// TIA Portal V20 export
// export: Created 2025-12-01T14:56:34.3256321Z, ExportSetting None, DisplayName Totally Integrated Automation Portal, DisplayVersion V20 Update 3, DisplayName TIA Portal Openness, DisplayVersion V20 Update 3, DisplayName TIA Portal Version Control Interface, DisplayVersion V20 Update 3, DisplayName STEP 7 Professional, DisplayVersion V20 Update 3, DisplayName STEP 7 Safety, DisplayVersion V20 Update 2, DisplayName WinCC Basic/Comfort/Advanced, DisplayVersion V20 Update 3, DisplayName WinCC Professional, DisplayVersion V20 Update 3, DisplayName WinCC Unified, DisplayVersion V20 Update 3
FUNCTION_BLOCK "FB463_CRTL_TR_TP_E1E2_S234_Pres"   // FB463, LAD
TITLE = bimba y lola
{ S7_Optimized_Access := 'FALSE' }
AUTHOR : TLigero
NAME : 20180827
VERSION : 3.0
// pendiente de simular
// stored: AutoNumber false, SetENOAutomatically false
   VAR_INPUT
      Mesa : UInt;   // Número de mesa
      En_Tension : Bool;
      pHsMx : Bool;   // pHs de presencia de la Mesa
      TP1_Up : Bool;   // TP1 Arriba. E1 >> S3. si no hay tope poner ON
      TP1_Down : Bool;   // TP1 Abajo. E1 >> S3. si no hay tope poner ON
      PosTR_E1 : Bool;   // Posicion del TR en E1E3
      PosTR_E2 : Bool;   // Posicion del TR en E2E4
      Termico_13 : Bool;   // Proteccion del Tx en E1E3
      Termico_24 : Bool;   // Proteccion del Tx en E2E4
      Avance_13 : Bool;   // Avance del Tx en E1E3
      Avance_24 : Bool;   // Avance del Tx en E2E4
      Retroceso_24 : Bool;   // Retroceso del Tx en E2E4
      PTF_Sal_M2 : Bool;   // S2 >> Mesa Siguiente PTF
      NXT_Avance_S2 : Bool;   // S2 >> Mesa Siguiente avanzando
      PTF_Sal_M3 : Bool;   // S3 >> Mesa Siguiente PTF
      NXT_Avance_S3 : Bool;   // S3 >> Mesa Siguiente avanzando
      PTF_Sal_M4 : Bool;   // S4 >> Mesa Siguiente PTF
      NXT_Avance_S4 : Bool;   // S4 >> Mesa Siguiente avanzando
      F_EnvMens_Mx : Bool;   // Fin de Envio de Mensaje
      Mx_Bloq_Activo : Bool;   // Bloqueo Activo de la Mesa
      Mx_FlujoPrin_S2 : Bool;   // para flujo principal S3 dejar los dos flujos principales a off
      Mx_FlujoPrin_S4 : Bool;   // para flujo principal S3 dejar los dos flujos principales a off
      AVTF_Ent_M1 : Bool;   // E1 >> Mesa Anterior AVTF
      AVTF_Ent_M2 : Bool;   // E2 >> Mesa Anterior AVTF
      Num_Cruce : UInt;   // Número de cruce.
      DB_FIFO_Cruce : UInt := 213;   // DB de la FIFO de ordenes del cruce
      Long_FIFO_Cruce : UInt := 1;   // Longitut de la FIFO de ordenes del cruce
      ValorOrden_S2 : Word := 16#81;   // Con que orden entra por S2
      ValorOrden_S4 : Word := 16#82;   // Con que orden entra por S4
      MesaS2 : UInt;   // Número de mesa por S2
      MesaS3 : UInt;   // Número de mesa por S3
      MesaS4 : UInt;   // Número de mesa por S4
      V_CNT_pHsMx_E1 : UDInt := 500;   // Valor de presencia por E1 en ms
      V_CNT_pHsMx_E2 : UDInt := 500;   // Valor de presencia por E2 en ms
      V_CNT_ApHsMx_S2 : UDInt := 500;   // Valor de Ausencia por S2 en ms
      V_CNT_ApHsMx_S3 : UDInt := 500;   // Valor de Ausencia por S3 en ms
      V_CNT_ApHsMx_S4 : UDInt := 500;   // Valor de Ausencia por S4 en ms
      V_TOut_Tx_Mx : UDInt := 3000;   // TimeOut de Atasco en ms
      V_TOut_TP : UDInt := 2000;   // TimeOut de Tope en ms
      V_TOut_TR : UDInt := 2000;   // TimeOut de Transfer en ms
      V_Paro : UDInt := 5000;   // tiempo que avanza el transportador sin aviso hasta que se para (ms)
      V_Vaciado : UDInt := 5000;   // Valor de vaciado en ms
   END_VAR
   VAR_OUTPUT
      P_EnvMens_PMx : Bool;   // Permiso de Enviar Mensaje de Presencia
      Etiqueta_Jdt : UDInt;   // Etiqueta que ha sido leida
      Orden_Ejecutada_Jdt : UInt;   // Orden que se ha ejecutado
      PTF_Ent_M1 : Bool;   // E1 >> Mesa Anterior PTF
      PTF_Ent_M2 : Bool;   // E2 >> Mesa Anterior PTF
      AVTF_Sal_M2 : Bool;   // S2 >> Mesa Siguiente AVTF
      NXT_Descarga_Act_S2 : Bool;   // S2 >> Mesa Siguiente descarga activa
      AVTF_Sal_M3 : Bool;   // S3 >> Mesa Siguiente AVTF
      NXT_Descarga_Act_S3 : Bool;   // S3 >> Mesa Siguiente descarga activa
      AVTF_Sal_M4 : Bool;   // S4 >> Mesa Siguiente AVTF
      NXT_Descarga_Act_S4 : Bool;   // S4 >> Mesa Siguiente descarga activa
   END_VAR
   VAR
      T1_ET00 : Bool;
      T1_ET01 : Bool;
      T1_ET02 : Bool;
      T1_ET03 : Bool;
      T1_ET10 : Bool;
      T1_ET11 : Bool;
      T1_ET20 : Bool;
      T1_ET21 : Bool;
      T1_ET50 : Bool;
      T1_ET60 : Bool;
      T1_ET80 : Bool;
      T1_ET110 : Bool;
      T1_ET111 : Bool;
      T1_ET112 : Bool;
      FIFO_OK : Bool;
      TRANS_OK : Bool;
      O_Bloqueo : Bool;
      Inv_sentido_24 : Bool;
      Ultima_entra_de_E2 : Bool;
      Ultima_entra_de_E1 : Bool;
      Err_Detec_PHS : Bool;
      Tim_Vaciado_Q : Bool;
      TMP_Atasco_Q : Bool;
      TMP_Paro_Q : Bool;
      FN_ET02 : Bool;
      Tmp_Tout_Tr_Q : Bool;
      TMP_Tout_tope_E2_Q : Bool;
      TMP_Tout_tope_E1_Q : Bool;
      maux_fp_disparo_e1 : Bool;
      maux_fp_disparo_e2 : Bool;
      TMP_pHs_E1 : UDInt;
      TMP_Aus_S2 : UDInt;
      TMP_Aus_S3 : UDInt;
      TMP_Aus_S4 : UDInt;
      CNT_pHs_E2 : UDInt;
      TIM_Vaciado : UDInt;
      TMP_Paro : UDInt;
      TMP_Tout_Tp_E2 : UDInt;
      TMP_Tout_Tp_E1 : UDInt;
      TMP_Tout_Tr : UDInt;
      TMP_Atasco : UDInt;
      TMP_En_tension : UDInt;
      Datos_Scanner { S7_SetPoint := 'True'} : "ROUT_Orden_Fifo_Scanner";
   END_VAR
   VAR_TEMP
      EstadoZona : "EstadoZona";   // Estado de Zona de la Mesa
      EstadoVI : "EstadosMesa";   // Estado del Vehiculo Inteliguente de la Mesa
      ConfigFB : "UDT_ConfigFB";   // Configuracion de la FB de la Mesa
      O_Sal_S2 : Bool;
      O_Sal_S4 : Bool;
      O_Sal_S3 : Bool;
      O_Vaciar : Bool;
      Moti_ERRO : Bool;
      Moti_NENC : Bool;
      Moti_NORM : Bool;
      Moti_INIC : Bool;
      tmp_Aus_S4_Q : Bool;
      tmp_pHs_E2_Q : Bool;
      tmp_pHs_E1_Q : Bool;
      tmp_pHs_S3_Q : Bool;
      tmp_pHs_S2_Q : Bool;
      ok_tension : Bool;
      Aux_W_Moti : Word;
      INT_ORDEN : UInt;
      Aux_W_Orden : Word;
      I_Ord_Filtrada : UInt;
      I_V_Ord_S4 : UInt;
      I_V_Ord_S2 : UInt;
   END_VAR
   VAR_TEMP   // added for the SCL form of the ladder/FBD networks
      _w1 : Bool;
      _w2 : Bool;
      _w3 : Bool;
      _w4 : Bool;
      _w5 : Bool;
      _w6 : Bool;
      _w7 : Bool;
   END_VAR
BEGIN

REGION Network 1: INICIALIZAR - Recoger las Variables de Estado de la Mesa
   // Se recoge - Estado_CBx
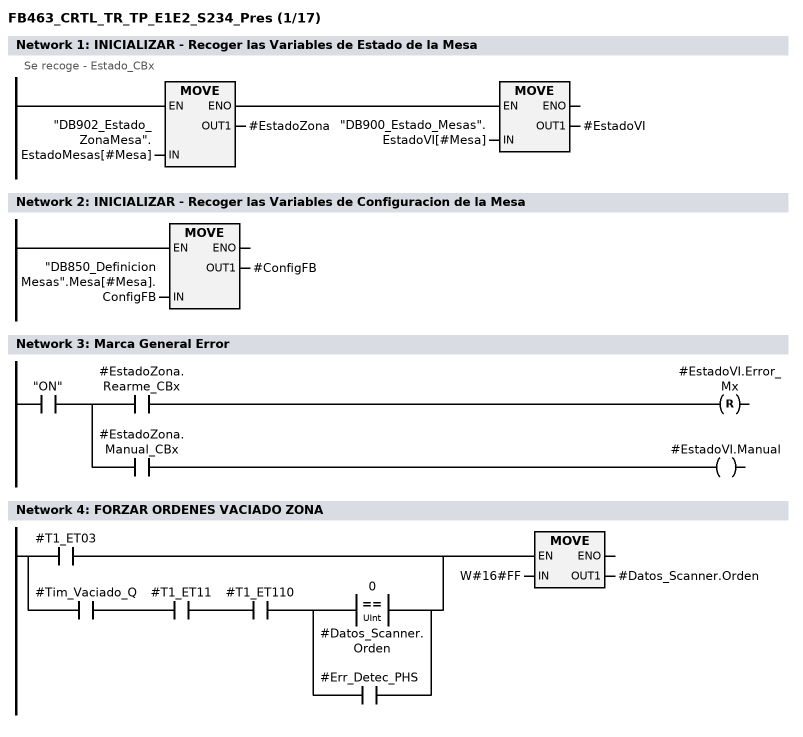
   RUNG wire#powerrail
      Move(in := "DB902_Estado_ZonaMesa".EstadoMesas[#Mesa], out1 => #EstadoZona)
      Move(in := "DB900_Estado_Mesas".EstadoVI[#Mesa], out1 => #EstadoVI)
   END_RUNG
   // the same network as SCL:
   #EstadoZona := "DB902_Estado_ZonaMesa".EstadoMesas[#Mesa];
   #EstadoVI := "DB900_Estado_Mesas".EstadoVI[#Mesa];
END_REGION

REGION Network 2: INICIALIZAR - Recoger las Variables de Configuracion de la Mesa
   RUNG wire#powerrail
      Move(in := "DB850_DefinicionMesas".Mesa[#Mesa].ConfigFB, out1 => #ConfigFB)
   END_RUNG
   // the same network as SCL:
   #ConfigFB := "DB850_DefinicionMesas".Mesa[#Mesa].ConfigFB;
END_REGION

REGION Network 3: Marca General Error
   RUNG wire#powerrail
      Contact( "ON" )
      wire#w1
      Contact( #EstadoZona.Rearme_CBx )
      R_Coil( #EstadoVI.Error_Mx )
   END_RUNG
   RUNG wire#w1
      Contact( #EstadoZona.Manual_CBx )
      Coil( #EstadoVI.Manual )
   END_RUNG
   // the same network as SCL:
   IF "ON" AND #EstadoZona.Rearme_CBx THEN #EstadoVI.Error_Mx := FALSE; END_IF;
   #EstadoVI.Manual := "ON" AND #EstadoZona.Manual_CBx;
END_REGION

REGION Network 4: FORZAR ORDENES VACIADO ZONA
   RUNG wire#powerrail
      Contact( #T1_ET03 )
      wire#w1
      { S7_GenerateENO := "TRUE" } Move(in := W#16#FF, out1 => #Datos_Scanner.Orden)
   END_RUNG
   RUNG wire#powerrail
      Contact( #Tim_Vaciado_Q )
      Contact( #T1_ET11 )
      Contact( #T1_ET110 )
      wire#w2
      { S7_Templates := "SrcType := UInt" } EQ_Contact(in1 := 0, in2 := #Datos_Scanner.Orden)
   END_RUNG wire#w1
   RUNG wire#w2
      Contact( #Err_Detec_PHS )
   END_RUNG wire#w1
   // the same network as SCL:
   IF #T1_ET03 OR (#Tim_Vaciado_Q AND #T1_ET11 AND #T1_ET110 AND ((0 = #Datos_Scanner.Orden) OR #Err_Detec_PHS)) THEN
       #Datos_Scanner.Orden := W#16#FF;
   END_IF;
END_REGION

REGION Network 5: evaluar la orden extraida de la fifo
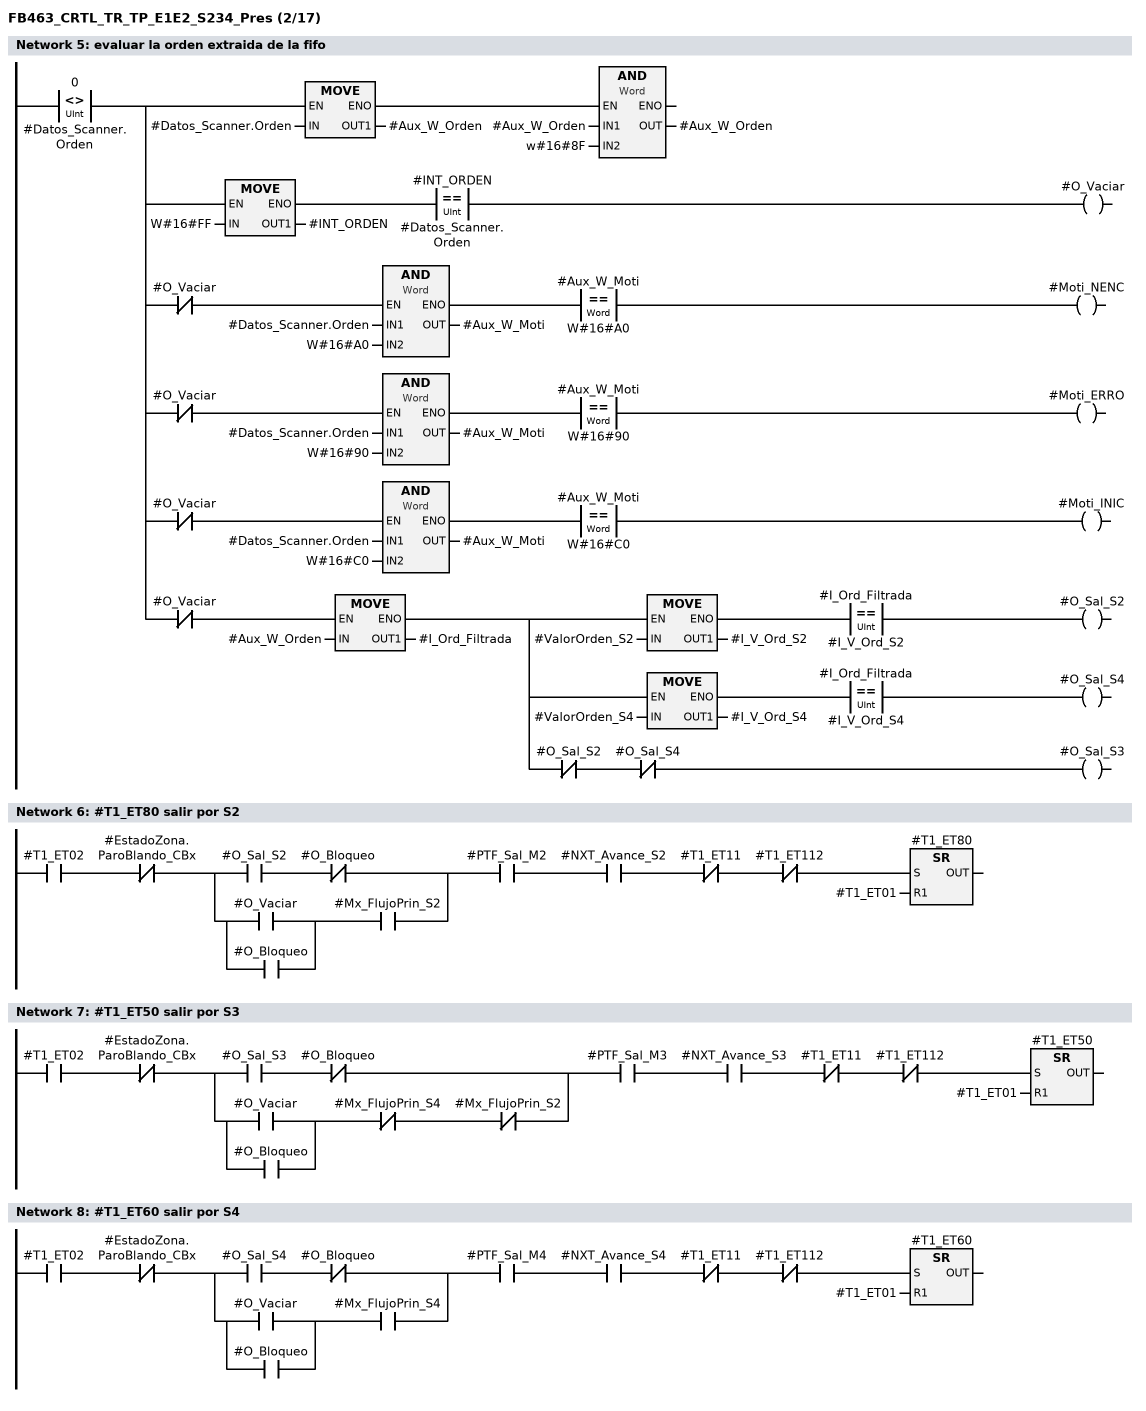
   RUNG wire#powerrail
      { S7_Templates := "SrcType := UInt" } NE_Contact(in1 := 0, in2 := #Datos_Scanner.Orden)
      wire#w1
      { S7_GenerateENO := "TRUE" } Move(in := #Datos_Scanner.Orden, out1 => #Aux_W_Orden)
      { S7_Templates := "SrcType := Word"; S7_GenerateENO := "TRUE" } And(in1 := #Aux_W_Orden, in2 := w#16#8F, out => #Aux_W_Orden)
   END_RUNG
   RUNG wire#w1
      { S7_GenerateENO := "TRUE" } Move(in := W#16#FF, out1 => #INT_ORDEN)
      { S7_Templates := "SrcType := UInt" } EQ_Contact(in1 := #INT_ORDEN, in2 := #Datos_Scanner.Orden)
      Coil( #O_Vaciar )
   END_RUNG
   RUNG wire#w1
      I_Contact( #O_Vaciar )
      { S7_Templates := "SrcType := Word"; S7_GenerateENO := "TRUE" } And(in1 := #Datos_Scanner.Orden, in2 := W#16#A0, out => #Aux_W_Moti)
      { S7_Templates := "SrcType := Word" } EQ_Contact(in1 := #Aux_W_Moti, in2 := W#16#A0)
      Coil( #Moti_NENC )
   END_RUNG
   RUNG wire#w1
      I_Contact( #O_Vaciar )
      { S7_Templates := "SrcType := Word"; S7_GenerateENO := "TRUE" } And(in1 := #Datos_Scanner.Orden, in2 := W#16#90, out => #Aux_W_Moti)
      { S7_Templates := "SrcType := Word" } EQ_Contact(in1 := #Aux_W_Moti, in2 := W#16#90)
      Coil( #Moti_ERRO )
   END_RUNG
   RUNG wire#w1
      I_Contact( #O_Vaciar )
      { S7_Templates := "SrcType := Word"; S7_GenerateENO := "TRUE" } And(in1 := #Datos_Scanner.Orden, in2 := W#16#C0, out => #Aux_W_Moti)
      { S7_Templates := "SrcType := Word" } EQ_Contact(in1 := #Aux_W_Moti, in2 := W#16#C0)
      Coil( #Moti_INIC )
   END_RUNG
   RUNG wire#w1
      I_Contact( #O_Vaciar )
      { S7_GenerateENO := "TRUE" } Move(in := #Aux_W_Orden, out1 => #I_Ord_Filtrada)
      wire#w2
      { S7_GenerateENO := "TRUE" } Move(in := #ValorOrden_S2, out1 => #I_V_Ord_S2)
      { S7_Templates := "SrcType := UInt" } EQ_Contact(in1 := #I_Ord_Filtrada, in2 := #I_V_Ord_S2)
      Coil( #O_Sal_S2 )
   END_RUNG
   RUNG wire#w2
      { S7_GenerateENO := "TRUE" } Move(in := #ValorOrden_S4, out1 => #I_V_Ord_S4)
      { S7_Templates := "SrcType := UInt" } EQ_Contact(in1 := #I_Ord_Filtrada, in2 := #I_V_Ord_S4)
      Coil( #O_Sal_S4 )
   END_RUNG
   RUNG wire#w2
      I_Contact( #O_Sal_S2 )
      I_Contact( #O_Sal_S4 )
      Coil( #O_Sal_S3 )
   END_RUNG
   // the same network as SCL:
   // ENO of a box is taken as its EN; it also drops when the box reports an error
   #_w1 := 0 <> #Datos_Scanner.Orden;
   IF #_w1 THEN
       #Aux_W_Orden := #Datos_Scanner.Orden;
       #Aux_W_Orden := #Aux_W_Orden AND w#16#8F;
       #INT_ORDEN := W#16#FF;
   END_IF;
   #O_Vaciar := #_w1 AND (#INT_ORDEN = #Datos_Scanner.Orden);
   #_w2 := #_w1 AND NOT #O_Vaciar;
   IF #_w2 THEN #Aux_W_Moti := #Datos_Scanner.Orden AND W#16#A0; END_IF;
   #Moti_NENC := #_w2 AND (#Aux_W_Moti = W#16#A0);
   #_w3 := #_w1 AND NOT #O_Vaciar;
   IF #_w3 THEN #Aux_W_Moti := #Datos_Scanner.Orden AND W#16#90; END_IF;
   #Moti_ERRO := #_w3 AND (#Aux_W_Moti = W#16#90);
   #_w4 := #_w1 AND NOT #O_Vaciar;
   IF #_w4 THEN #Aux_W_Moti := #Datos_Scanner.Orden AND W#16#C0; END_IF;
   #Moti_INIC := #_w4 AND (#Aux_W_Moti = W#16#C0);
   #_w5 := #_w1 AND NOT #O_Vaciar;
   IF #_w5 THEN
       #I_Ord_Filtrada := #Aux_W_Orden;
       #I_V_Ord_S2 := #ValorOrden_S2;
   END_IF;
   #O_Sal_S2 := #_w5 AND (#I_Ord_Filtrada = #I_V_Ord_S2);
   IF #_w5 THEN #I_V_Ord_S4 := #ValorOrden_S4; END_IF;
   #O_Sal_S4 := #_w5 AND (#I_Ord_Filtrada = #I_V_Ord_S4);
   #O_Sal_S3 := #_w5 AND NOT #O_Sal_S2 AND NOT #O_Sal_S4;
END_REGION

REGION Network 6: #T1_ET80 salir por S2
   RUNG wire#powerrail
      Contact( #T1_ET02 )
      I_Contact( #EstadoZona.ParoBlando_CBx )
      wire#w1
      Contact( #O_Sal_S2 )
      I_Contact( #O_Bloqueo )
      wire#w2
      Contact( #PTF_Sal_M2 )
      Contact( #NXT_Avance_S2 )
      I_Contact( #T1_ET11 )
      I_Contact( #T1_ET112 )
      S_SR(operand := #T1_ET80, r1 := #T1_ET01)
   END_RUNG
   RUNG wire#w1
      Contact( #O_Vaciar )
      wire#w3
      Contact( #Mx_FlujoPrin_S2 )
   END_RUNG wire#w2
   RUNG wire#w1
      Contact( #O_Bloqueo )
   END_RUNG wire#w3
   // the same network as SCL:
   IF #T1_ET02 AND NOT #EstadoZona.ParoBlando_CBx AND ((#O_Sal_S2 AND NOT #O_Bloqueo) OR ((#O_Vaciar OR #O_Bloqueo) AND #Mx_FlujoPrin_S2)) AND #PTF_Sal_M2 AND #NXT_Avance_S2 AND NOT #T1_ET11 AND NOT #T1_ET112 THEN
       #T1_ET80 := TRUE;   // SR flip-flop
   END_IF;
   IF #T1_ET01 THEN #T1_ET80 := FALSE; END_IF;
END_REGION

REGION Network 7: #T1_ET50 salir por S3
   RUNG wire#powerrail
      Contact( #T1_ET02 )
      I_Contact( #EstadoZona.ParoBlando_CBx )
      wire#w1
      Contact( #O_Sal_S3 )
      I_Contact( #O_Bloqueo )
      wire#w2
      Contact( #PTF_Sal_M3 )
      Contact( #NXT_Avance_S3 )
      I_Contact( #T1_ET11 )
      I_Contact( #T1_ET112 )
      S_SR(operand := #T1_ET50, r1 := #T1_ET01)
   END_RUNG
   RUNG wire#w1
      Contact( #O_Vaciar )
      wire#w3
      I_Contact( #Mx_FlujoPrin_S4 )
      I_Contact( #Mx_FlujoPrin_S2 )
   END_RUNG wire#w2
   RUNG wire#w1
      Contact( #O_Bloqueo )
   END_RUNG wire#w3
   // the same network as SCL:
   IF #T1_ET02 AND NOT #EstadoZona.ParoBlando_CBx AND ((#O_Sal_S3 AND NOT #O_Bloqueo) OR ((#O_Vaciar OR #O_Bloqueo) AND NOT #Mx_FlujoPrin_S4 AND NOT #Mx_FlujoPrin_S2)) AND #PTF_Sal_M3 AND #NXT_Avance_S3 AND NOT #T1_ET11 AND NOT #T1_ET112 THEN
       #T1_ET50 := TRUE;   // SR flip-flop
   END_IF;
   IF #T1_ET01 THEN #T1_ET50 := FALSE; END_IF;
END_REGION

REGION Network 8: #T1_ET60 salir por S4
   RUNG wire#powerrail
      Contact( #T1_ET02 )
      I_Contact( #EstadoZona.ParoBlando_CBx )
      wire#w1
      Contact( #O_Sal_S4 )
      I_Contact( #O_Bloqueo )
      wire#w2
      Contact( #PTF_Sal_M4 )
      Contact( #NXT_Avance_S4 )
      I_Contact( #T1_ET11 )
      I_Contact( #T1_ET112 )
      S_SR(operand := #T1_ET60, r1 := #T1_ET01)
   END_RUNG
   RUNG wire#w1
      Contact( #O_Vaciar )
      wire#w3
      Contact( #Mx_FlujoPrin_S4 )
   END_RUNG wire#w2
   RUNG wire#w1
      Contact( #O_Bloqueo )
   END_RUNG wire#w3
   // the same network as SCL:
   IF #T1_ET02 AND NOT #EstadoZona.ParoBlando_CBx AND ((#O_Sal_S4 AND NOT #O_Bloqueo) OR ((#O_Vaciar OR #O_Bloqueo) AND #Mx_FlujoPrin_S4)) AND #PTF_Sal_M4 AND #NXT_Avance_S4 AND NOT #T1_ET11 AND NOT #T1_ET112 THEN
       #T1_ET60 := TRUE;   // SR flip-flop
   END_IF;
   IF #T1_ET01 THEN #T1_ET60 := FALSE; END_IF;
END_REGION

REGION Network 9: #T1_ET02. ESTADO REPOSO CARGADA.
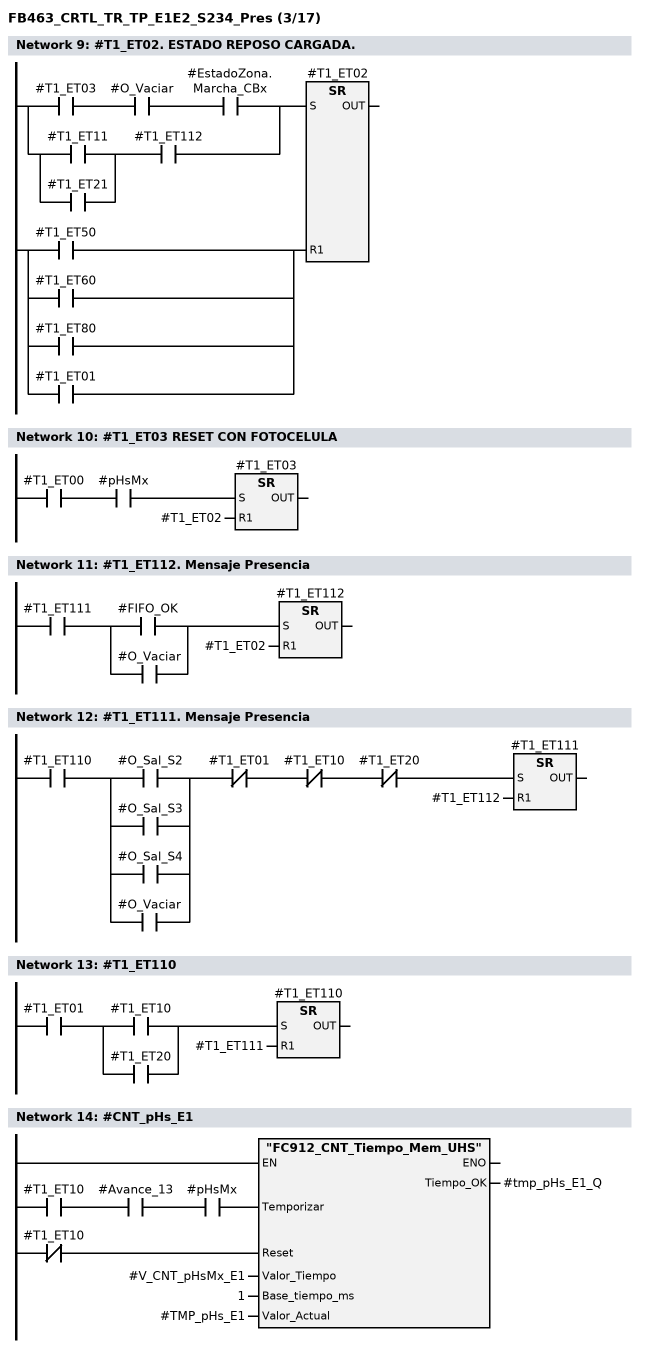
   RUNG wire#powerrail
      Contact( #T1_ET03 )
      Contact( #O_Vaciar )
      Contact( #EstadoZona.Marcha_CBx )
      wire#w1
      S_SR(operand := #T1_ET02, r1 := wire#w3)
   END_RUNG
   RUNG wire#powerrail
      Contact( #T1_ET11 )
      wire#w2
      Contact( #T1_ET112 )
   END_RUNG wire#w1
   RUNG wire#powerrail
      Contact( #T1_ET21 )
   END_RUNG wire#w2
   RUNG wire#powerrail
      Contact( #T1_ET50 )
   END_RUNG wire#w3
   RUNG wire#powerrail
      Contact( #T1_ET60 )
   END_RUNG wire#w3
   RUNG wire#powerrail
      Contact( #T1_ET80 )
   END_RUNG wire#w3
   RUNG wire#powerrail
      Contact( #T1_ET01 )
   END_RUNG wire#w3
   // the same network as SCL:
   IF (#T1_ET03 AND #O_Vaciar AND #EstadoZona.Marcha_CBx) OR ((#T1_ET11 OR #T1_ET21) AND #T1_ET112) THEN
       #T1_ET02 := TRUE;   // SR flip-flop
   END_IF;
   IF #T1_ET50 OR #T1_ET60 OR #T1_ET80 OR #T1_ET01 THEN #T1_ET02 := FALSE; END_IF;
END_REGION

REGION Network 10: #T1_ET03 RESET CON FOTOCELULA
   RUNG wire#powerrail
      Contact( #T1_ET00 )
      Contact( #pHsMx )
      S_SR(operand := #T1_ET03, r1 := #T1_ET02)
   END_RUNG
   // the same network as SCL:
   IF #T1_ET00 AND #pHsMx THEN
       #T1_ET03 := TRUE;   // SR flip-flop
   END_IF;
   IF #T1_ET02 THEN #T1_ET03 := FALSE; END_IF;
END_REGION

REGION Network 11: #T1_ET112. Mensaje Presencia
   RUNG wire#powerrail
      Contact( #T1_ET111 )
      wire#w1
      Contact( #FIFO_OK )
      wire#w2
      S_SR(operand := #T1_ET112, r1 := #T1_ET02)
   END_RUNG
   RUNG wire#w1
      Contact( #O_Vaciar )
   END_RUNG wire#w2
   // the same network as SCL:
   IF #T1_ET111 AND (#FIFO_OK OR #O_Vaciar) THEN
       #T1_ET112 := TRUE;   // SR flip-flop
   END_IF;
   IF #T1_ET02 THEN #T1_ET112 := FALSE; END_IF;
END_REGION

REGION Network 12: #T1_ET111. Mensaje Presencia
   RUNG wire#powerrail
      Contact( #T1_ET110 )
      wire#w1
      Contact( #O_Sal_S2 )
      wire#w2
      I_Contact( #T1_ET01 )
      I_Contact( #T1_ET10 )
      I_Contact( #T1_ET20 )
      S_SR(operand := #T1_ET111, r1 := #T1_ET112)
   END_RUNG
   RUNG wire#w1
      Contact( #O_Sal_S3 )
   END_RUNG wire#w2
   RUNG wire#w1
      Contact( #O_Sal_S4 )
   END_RUNG wire#w2
   RUNG wire#w1
      Contact( #O_Vaciar )
   END_RUNG wire#w2
   // the same network as SCL:
   IF #T1_ET110 AND (#O_Sal_S2 OR #O_Sal_S3 OR #O_Sal_S4 OR #O_Vaciar) AND NOT #T1_ET01 AND NOT #T1_ET10 AND NOT #T1_ET20 THEN
       #T1_ET111 := TRUE;   // SR flip-flop
   END_IF;
   IF #T1_ET112 THEN #T1_ET111 := FALSE; END_IF;
END_REGION

REGION Network 13: #T1_ET110
   RUNG wire#powerrail
      Contact( #T1_ET01 )
      wire#w1
      Contact( #T1_ET10 )
      wire#w2
      S_SR(operand := #T1_ET110, r1 := #T1_ET111)
   END_RUNG
   RUNG wire#w1
      Contact( #T1_ET20 )
   END_RUNG wire#w2
   // the same network as SCL:
   IF #T1_ET01 AND (#T1_ET10 OR #T1_ET20) THEN
       #T1_ET110 := TRUE;   // SR flip-flop
   END_IF;
   IF #T1_ET111 THEN #T1_ET110 := FALSE; END_IF;
END_REGION

REGION Network 14: #CNT_pHs_E1
   RUNG wire#powerrail
      "FC912_CNT_Tiempo_Mem_UHS"(Temporizar := wire#w1, Reset := wire#w2, Valor_Tiempo := #V_CNT_pHsMx_E1, Base_tiempo_ms := 1, Valor_Actual := #TMP_pHs_E1, Tiempo_OK => #tmp_pHs_E1_Q)
   END_RUNG
   RUNG wire#powerrail
      Contact( #T1_ET10 )
      Contact( #Avance_13 )
      Contact( #pHsMx )
   END_RUNG wire#w1
   RUNG wire#powerrail
      I_Contact( #T1_ET10 )
   END_RUNG wire#w2
   // the same network as SCL:
   "FC912_CNT_Tiempo_Mem_UHS"(Temporizar := #T1_ET10 AND #Avance_13 AND #pHsMx,
                           Reset := NOT #T1_ET10,
                           Valor_Tiempo := #V_CNT_pHsMx_E1,
                           Base_tiempo_ms := 1,
                           Valor_Actual := #TMP_pHs_E1,
                           Tiempo_OK => #tmp_pHs_E1_Q);
END_REGION

REGION Network 15: #CNT_pHs_E2
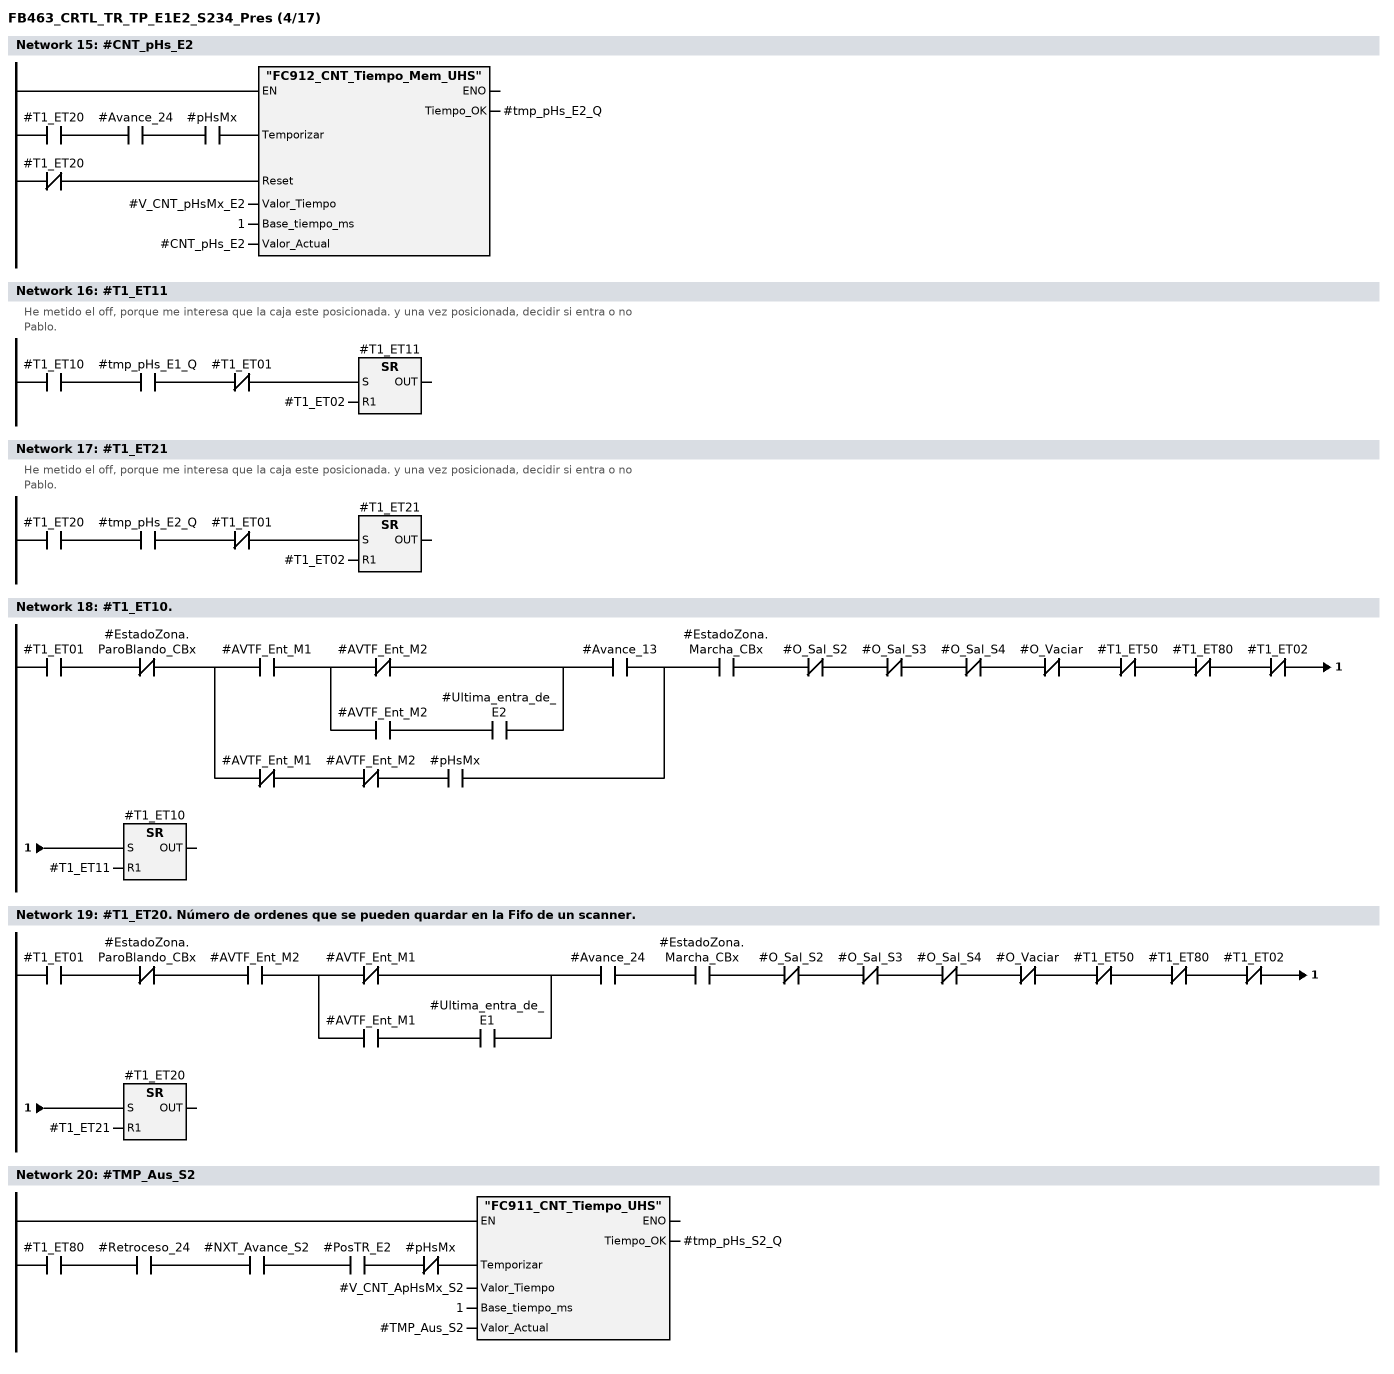
   RUNG wire#powerrail
      "FC912_CNT_Tiempo_Mem_UHS"(Temporizar := wire#w1, Reset := wire#w2, Valor_Tiempo := #V_CNT_pHsMx_E2, Base_tiempo_ms := 1, Valor_Actual := #CNT_pHs_E2, Tiempo_OK => #tmp_pHs_E2_Q)
   END_RUNG
   RUNG wire#powerrail
      Contact( #T1_ET20 )
      Contact( #Avance_24 )
      Contact( #pHsMx )
   END_RUNG wire#w1
   RUNG wire#powerrail
      I_Contact( #T1_ET20 )
   END_RUNG wire#w2
   // the same network as SCL:
   "FC912_CNT_Tiempo_Mem_UHS"(Temporizar := #T1_ET20 AND #Avance_24 AND #pHsMx,
                           Reset := NOT #T1_ET20,
                           Valor_Tiempo := #V_CNT_pHsMx_E2,
                           Base_tiempo_ms := 1,
                           Valor_Actual := #CNT_pHs_E2,
                           Tiempo_OK => #tmp_pHs_E2_Q);
END_REGION

REGION Network 16: #T1_ET11
   // He metido el off, porque me interesa que la caja este posicionada. y una vez posicionada, decidir si entra o no
   // Pablo.
   RUNG wire#powerrail
      Contact( #T1_ET10 )
      Contact( #tmp_pHs_E1_Q )
      I_Contact( #T1_ET01 )
      S_SR(operand := #T1_ET11, r1 := #T1_ET02)
   END_RUNG
   // the same network as SCL:
   IF #T1_ET10 AND #tmp_pHs_E1_Q AND NOT #T1_ET01 THEN
       #T1_ET11 := TRUE;   // SR flip-flop
   END_IF;
   IF #T1_ET02 THEN #T1_ET11 := FALSE; END_IF;
END_REGION

REGION Network 17: #T1_ET21
   // He metido el off, porque me interesa que la caja este posicionada. y una vez posicionada, decidir si entra o no
   // Pablo.
   RUNG wire#powerrail
      Contact( #T1_ET20 )
      Contact( #tmp_pHs_E2_Q )
      I_Contact( #T1_ET01 )
      S_SR(operand := #T1_ET21, r1 := #T1_ET02)
   END_RUNG
   // the same network as SCL:
   IF #T1_ET20 AND #tmp_pHs_E2_Q AND NOT #T1_ET01 THEN
       #T1_ET21 := TRUE;   // SR flip-flop
   END_IF;
   IF #T1_ET02 THEN #T1_ET21 := FALSE; END_IF;
END_REGION

REGION Network 18: #T1_ET10.
   RUNG wire#powerrail
      Contact( #T1_ET01 )
      I_Contact( #EstadoZona.ParoBlando_CBx )
      wire#w1
      Contact( #AVTF_Ent_M1 )
      wire#w2
      I_Contact( #AVTF_Ent_M2 )
      wire#w3
      Contact( #Avance_13 )
      wire#w4
      Contact( #EstadoZona.Marcha_CBx )
      I_Contact( #O_Sal_S2 )
      I_Contact( #O_Sal_S3 )
      I_Contact( #O_Sal_S4 )
      I_Contact( #O_Vaciar )
      I_Contact( #T1_ET50 )
      I_Contact( #T1_ET80 )
      I_Contact( #T1_ET02 )
      S_SR(operand := #T1_ET10, r1 := #T1_ET11)
   END_RUNG
   RUNG wire#w2
      Contact( #AVTF_Ent_M2 )
      Contact( #Ultima_entra_de_E2 )
   END_RUNG wire#w3
   RUNG wire#w1
      I_Contact( #AVTF_Ent_M1 )
      I_Contact( #AVTF_Ent_M2 )
      Contact( #pHsMx )
   END_RUNG wire#w4
   // the same network as SCL:
   IF #T1_ET01 AND NOT #EstadoZona.ParoBlando_CBx AND ((#AVTF_Ent_M1 AND (NOT #AVTF_Ent_M2 OR (#AVTF_Ent_M2 AND #Ultima_entra_de_E2)) AND #Avance_13) OR (NOT #AVTF_Ent_M1 AND NOT #AVTF_Ent_M2 AND #pHsMx)) AND #EstadoZona.Marcha_CBx AND NOT #O_Sal_S2 AND NOT #O_Sal_S3 AND NOT #O_Sal_S4 AND NOT #O_Vaciar AND NOT #T1_ET50 AND NOT #T1_ET80 AND NOT #T1_ET02 THEN
       #T1_ET10 := TRUE;   // SR flip-flop
   END_IF;
   IF #T1_ET11 THEN #T1_ET10 := FALSE; END_IF;
END_REGION

REGION Network 19: #T1_ET20. Número de ordenes que se pueden quardar en la Fifo de un scanner.
   RUNG wire#powerrail
      Contact( #T1_ET01 )
      I_Contact( #EstadoZona.ParoBlando_CBx )
      Contact( #AVTF_Ent_M2 )
      wire#w1
      I_Contact( #AVTF_Ent_M1 )
      wire#w2
      Contact( #Avance_24 )
      Contact( #EstadoZona.Marcha_CBx )
      I_Contact( #O_Sal_S2 )
      I_Contact( #O_Sal_S3 )
      I_Contact( #O_Sal_S4 )
      I_Contact( #O_Vaciar )
      I_Contact( #T1_ET50 )
      I_Contact( #T1_ET80 )
      I_Contact( #T1_ET02 )
      S_SR(operand := #T1_ET20, r1 := #T1_ET21)
   END_RUNG
   RUNG wire#w1
      Contact( #AVTF_Ent_M1 )
      Contact( #Ultima_entra_de_E1 )
   END_RUNG wire#w2
   // the same network as SCL:
   IF #T1_ET01 AND NOT #EstadoZona.ParoBlando_CBx AND #AVTF_Ent_M2 AND (NOT #AVTF_Ent_M1 OR (#AVTF_Ent_M1 AND #Ultima_entra_de_E1)) AND #Avance_24 AND #EstadoZona.Marcha_CBx AND NOT #O_Sal_S2 AND NOT #O_Sal_S3 AND NOT #O_Sal_S4 AND NOT #O_Vaciar AND NOT #T1_ET50 AND NOT #T1_ET80 AND NOT #T1_ET02 THEN
       #T1_ET20 := TRUE;   // SR flip-flop
   END_IF;
   IF #T1_ET21 THEN #T1_ET20 := FALSE; END_IF;
END_REGION

REGION Network 20: #TMP_Aus_S2
   RUNG wire#powerrail
      "FC911_CNT_Tiempo_UHS"(Temporizar := wire#w1, Valor_Tiempo := #V_CNT_ApHsMx_S2, Base_tiempo_ms := 1, Valor_Actual := #TMP_Aus_S2, Tiempo_OK => #tmp_pHs_S2_Q)
   END_RUNG
   RUNG wire#powerrail
      Contact( #T1_ET80 )
      Contact( #Retroceso_24 )
      Contact( #NXT_Avance_S2 )
      Contact( #PosTR_E2 )
      I_Contact( #pHsMx )
   END_RUNG wire#w1
   // the same network as SCL:
   "FC911_CNT_Tiempo_UHS"(Temporizar := #T1_ET80 AND #Retroceso_24 AND #NXT_Avance_S2 AND #PosTR_E2 AND NOT #pHsMx,
                          Valor_Tiempo := #V_CNT_ApHsMx_S2,
                          Base_tiempo_ms := 1,
                          Valor_Actual := #TMP_Aus_S2,
                          Tiempo_OK => #tmp_pHs_S2_Q);
END_REGION

REGION Network 21: #TMP_Aus_S3
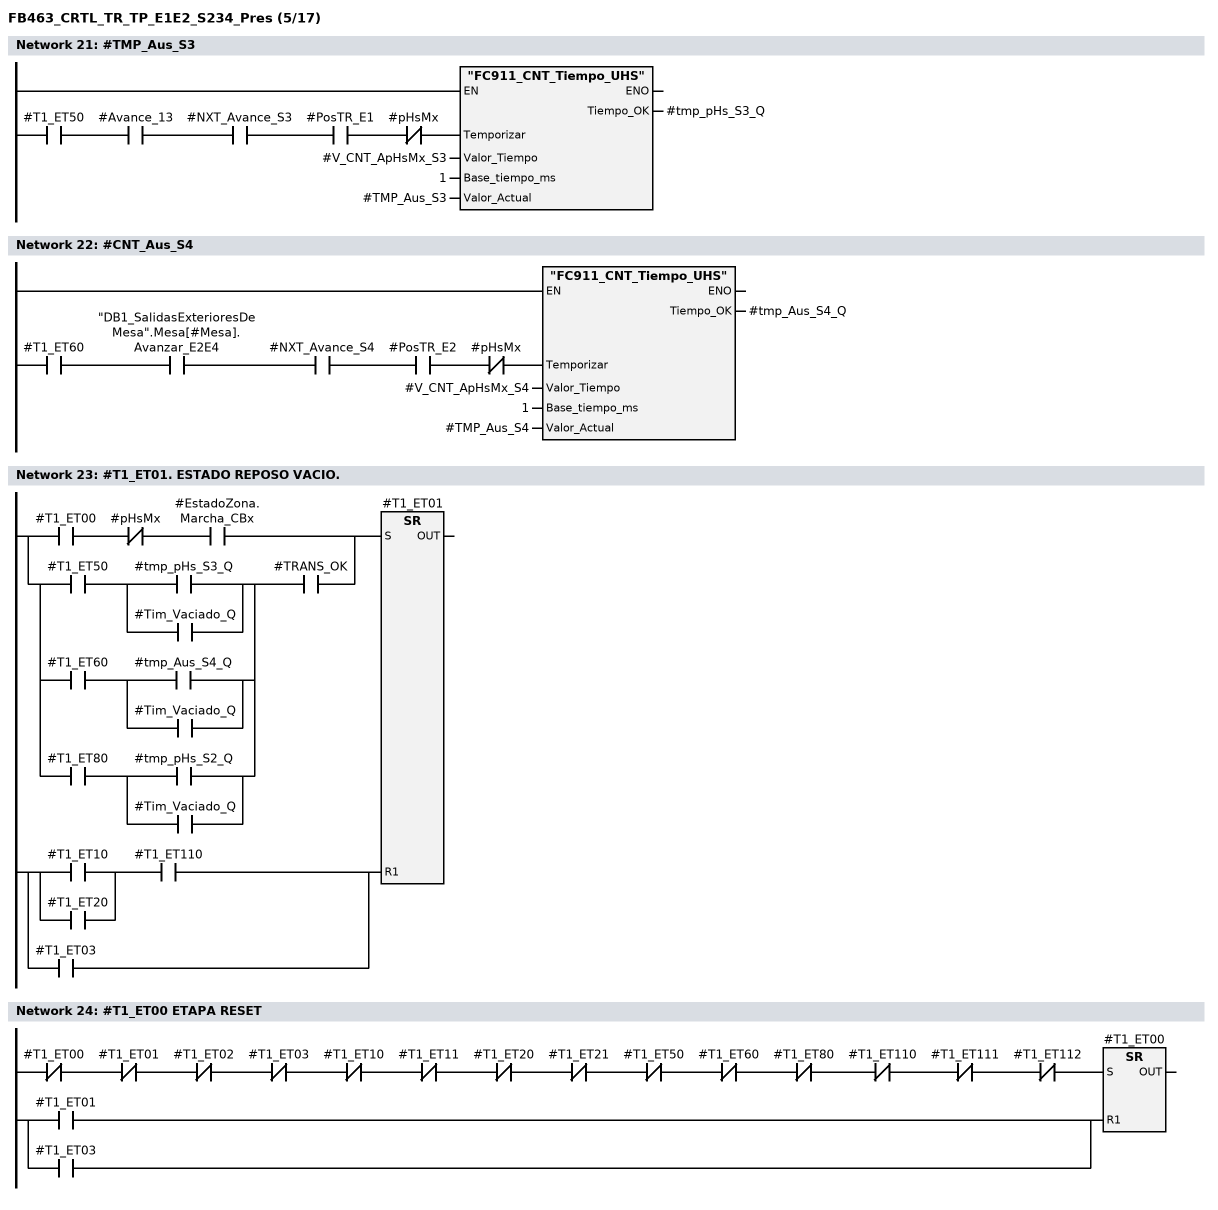
   RUNG wire#powerrail
      "FC911_CNT_Tiempo_UHS"(Temporizar := wire#w1, Valor_Tiempo := #V_CNT_ApHsMx_S3, Base_tiempo_ms := 1, Valor_Actual := #TMP_Aus_S3, Tiempo_OK => #tmp_pHs_S3_Q)
   END_RUNG
   RUNG wire#powerrail
      Contact( #T1_ET50 )
      Contact( #Avance_13 )
      Contact( #NXT_Avance_S3 )
      Contact( #PosTR_E1 )
      I_Contact( #pHsMx )
   END_RUNG wire#w1
   // the same network as SCL:
   "FC911_CNT_Tiempo_UHS"(Temporizar := #T1_ET50 AND #Avance_13 AND #NXT_Avance_S3 AND #PosTR_E1 AND NOT #pHsMx,
                          Valor_Tiempo := #V_CNT_ApHsMx_S3,
                          Base_tiempo_ms := 1,
                          Valor_Actual := #TMP_Aus_S3,
                          Tiempo_OK => #tmp_pHs_S3_Q);
END_REGION

REGION Network 22: #CNT_Aus_S4
   RUNG wire#powerrail
      "FC911_CNT_Tiempo_UHS"(Temporizar := wire#w1, Valor_Tiempo := #V_CNT_ApHsMx_S4, Base_tiempo_ms := 1, Valor_Actual := #TMP_Aus_S4, Tiempo_OK => #tmp_Aus_S4_Q)
   END_RUNG
   RUNG wire#powerrail
      Contact( #T1_ET60 )
      Contact( "DB1_SalidasExterioresDeMesa".Mesa[#Mesa].Avanzar_E2E4 )
      Contact( #NXT_Avance_S4 )
      Contact( #PosTR_E2 )
      I_Contact( #pHsMx )
   END_RUNG wire#w1
   // the same network as SCL:
   "FC911_CNT_Tiempo_UHS"(Temporizar := #T1_ET60 AND "DB1_SalidasExterioresDeMesa".Mesa[#Mesa].Avanzar_E2E4 AND #NXT_Avance_S4 AND #PosTR_E2 AND NOT #pHsMx,
                          Valor_Tiempo := #V_CNT_ApHsMx_S4,
                          Base_tiempo_ms := 1,
                          Valor_Actual := #TMP_Aus_S4,
                          Tiempo_OK => #tmp_Aus_S4_Q);
END_REGION

REGION Network 23: #T1_ET01. ESTADO REPOSO VACIO.
   RUNG wire#powerrail
      Contact( #T1_ET00 )
      I_Contact( #pHsMx )
      Contact( #EstadoZona.Marcha_CBx )
      wire#w1
      S_SR(operand := #T1_ET01, r1 := wire#w7)
   END_RUNG
   RUNG wire#powerrail
      Contact( #T1_ET50 )
      wire#w2
      Contact( #tmp_pHs_S3_Q )
      wire#w3
      Contact( #TRANS_OK )
   END_RUNG wire#w1
   RUNG wire#w2
      Contact( #Tim_Vaciado_Q )
   END_RUNG wire#w3
   RUNG wire#powerrail
      Contact( #T1_ET60 )
      wire#w4
      Contact( #tmp_Aus_S4_Q )
   END_RUNG wire#w3
   RUNG wire#w4
      Contact( #Tim_Vaciado_Q )
   END_RUNG wire#w3
   RUNG wire#powerrail
      Contact( #T1_ET80 )
      wire#w5
      Contact( #tmp_pHs_S2_Q )
   END_RUNG wire#w3
   RUNG wire#w5
      Contact( #Tim_Vaciado_Q )
   END_RUNG wire#w3
   RUNG wire#powerrail
      Contact( #T1_ET10 )
      wire#w6
      Contact( #T1_ET110 )
   END_RUNG wire#w7
   RUNG wire#powerrail
      Contact( #T1_ET20 )
   END_RUNG wire#w6
   RUNG wire#powerrail
      Contact( #T1_ET03 )
   END_RUNG wire#w7
   // the same network as SCL:
   IF (#T1_ET00 AND NOT #pHsMx AND #EstadoZona.Marcha_CBx) OR (((#T1_ET50 AND (#tmp_pHs_S3_Q OR #Tim_Vaciado_Q)) OR (#T1_ET60 AND (#tmp_Aus_S4_Q OR #Tim_Vaciado_Q)) OR (#T1_ET80 AND (#tmp_pHs_S2_Q OR #Tim_Vaciado_Q))) AND #TRANS_OK) THEN
       #T1_ET01 := TRUE;   // SR flip-flop
   END_IF;
   IF ((#T1_ET10 OR #T1_ET20) AND #T1_ET110) OR #T1_ET03 THEN #T1_ET01 := FALSE; END_IF;
END_REGION

REGION Network 24: #T1_ET00 ETAPA RESET
   RUNG wire#powerrail
      I_Contact( #T1_ET00 )
      I_Contact( #T1_ET01 )
      I_Contact( #T1_ET02 )
      I_Contact( #T1_ET03 )
      I_Contact( #T1_ET10 )
      I_Contact( #T1_ET11 )
      I_Contact( #T1_ET20 )
      I_Contact( #T1_ET21 )
      I_Contact( #T1_ET50 )
      I_Contact( #T1_ET60 )
      I_Contact( #T1_ET80 )
      I_Contact( #T1_ET110 )
      I_Contact( #T1_ET111 )
      I_Contact( #T1_ET112 )
      S_SR(operand := #T1_ET00, r1 := wire#w1)
   END_RUNG
   RUNG wire#powerrail
      Contact( #T1_ET01 )
   END_RUNG wire#w1
   RUNG wire#powerrail
      Contact( #T1_ET03 )
   END_RUNG wire#w1
   // the same network as SCL:
   IF NOT #T1_ET00 AND NOT #T1_ET01 AND NOT #T1_ET02 AND NOT #T1_ET03 AND NOT #T1_ET10 AND NOT #T1_ET11 AND NOT #T1_ET20 AND NOT #T1_ET21 AND NOT #T1_ET50 AND NOT #T1_ET60 AND NOT #T1_ET80 AND NOT #T1_ET110 AND NOT #T1_ET111 AND NOT #T1_ET112 THEN
       #T1_ET00 := TRUE;   // SR flip-flop
   END_IF;
   IF #T1_ET01 OR #T1_ET03 THEN #T1_ET00 := FALSE; END_IF;
END_REGION

REGION Network 25: #TMP_Err_Subir_Tp
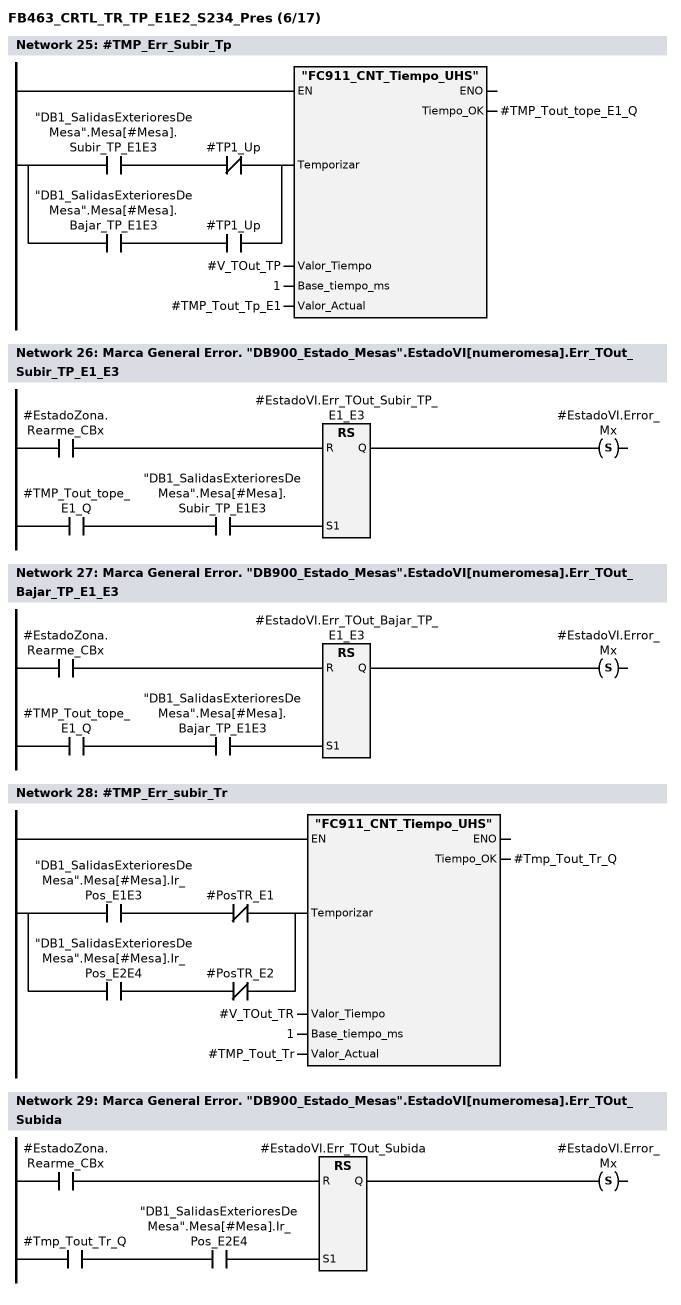
   RUNG wire#powerrail
      "FC911_CNT_Tiempo_UHS"(Temporizar := wire#w1, Valor_Tiempo := #V_TOut_TP, Base_tiempo_ms := 1, Valor_Actual := #TMP_Tout_Tp_E1, Tiempo_OK => #TMP_Tout_tope_E1_Q)
   END_RUNG
   RUNG wire#powerrail
      Contact( "DB1_SalidasExterioresDeMesa".Mesa[#Mesa].Subir_TP_E1E3 )
      I_Contact( #TP1_Up )
   END_RUNG wire#w1
   RUNG wire#powerrail
      Contact( "DB1_SalidasExterioresDeMesa".Mesa[#Mesa].Bajar_TP_E1E3 )
      Contact( #TP1_Up )
   END_RUNG wire#w1
   // the same network as SCL:
   "FC911_CNT_Tiempo_UHS"(Temporizar := ("DB1_SalidasExterioresDeMesa".Mesa[#Mesa].Subir_TP_E1E3 AND NOT #TP1_Up) OR ("DB1_SalidasExterioresDeMesa".Mesa[#Mesa].Bajar_TP_E1E3 AND #TP1_Up),
                          Valor_Tiempo := #V_TOut_TP,
                          Base_tiempo_ms := 1,
                          Valor_Actual := #TMP_Tout_Tp_E1,
                          Tiempo_OK => #TMP_Tout_tope_E1_Q);
END_REGION

REGION Network 26: Marca General Error. "DB900_Estado_Mesas".EstadoVI[numeromesa].Err_TOut_Subir_TP_E1_E3
   RUNG wire#powerrail
      Contact( #EstadoZona.Rearme_CBx )
      S_RS(operand := #EstadoVI.Err_TOut_Subir_TP_E1_E3, s1 := wire#w1)
      S_Coil( #EstadoVI.Error_Mx )
   END_RUNG
   RUNG wire#powerrail
      Contact( #TMP_Tout_tope_E1_Q )
      Contact( "DB1_SalidasExterioresDeMesa".Mesa[#Mesa].Subir_TP_E1E3 )
   END_RUNG wire#w1
   // the same network as SCL:
   IF #EstadoZona.Rearme_CBx THEN
       #EstadoVI.Err_TOut_Subir_TP_E1_E3 := FALSE;   // RS flip-flop
   END_IF;
   IF #TMP_Tout_tope_E1_Q AND "DB1_SalidasExterioresDeMesa".Mesa[#Mesa].Subir_TP_E1E3 THEN
       #EstadoVI.Err_TOut_Subir_TP_E1_E3 := TRUE;
   END_IF;
   IF #EstadoVI.Err_TOut_Subir_TP_E1_E3 THEN #EstadoVI.Error_Mx := TRUE; END_IF;
END_REGION

REGION Network 27: Marca General Error. "DB900_Estado_Mesas".EstadoVI[numeromesa].Err_TOut_Bajar_TP_E1_E3
   RUNG wire#powerrail
      Contact( #EstadoZona.Rearme_CBx )
      S_RS(operand := #EstadoVI.Err_TOut_Bajar_TP_E1_E3, s1 := wire#w1)
      S_Coil( #EstadoVI.Error_Mx )
   END_RUNG
   RUNG wire#powerrail
      Contact( #TMP_Tout_tope_E1_Q )
      Contact( "DB1_SalidasExterioresDeMesa".Mesa[#Mesa].Bajar_TP_E1E3 )
   END_RUNG wire#w1
   // the same network as SCL:
   IF #EstadoZona.Rearme_CBx THEN
       #EstadoVI.Err_TOut_Bajar_TP_E1_E3 := FALSE;   // RS flip-flop
   END_IF;
   IF #TMP_Tout_tope_E1_Q AND "DB1_SalidasExterioresDeMesa".Mesa[#Mesa].Bajar_TP_E1E3 THEN
       #EstadoVI.Err_TOut_Bajar_TP_E1_E3 := TRUE;
   END_IF;
   IF #EstadoVI.Err_TOut_Bajar_TP_E1_E3 THEN #EstadoVI.Error_Mx := TRUE; END_IF;
END_REGION

REGION Network 28: #TMP_Err_subir_Tr
   RUNG wire#powerrail
      "FC911_CNT_Tiempo_UHS"(Temporizar := wire#w1, Valor_Tiempo := #V_TOut_TR, Base_tiempo_ms := 1, Valor_Actual := #TMP_Tout_Tr, Tiempo_OK => #Tmp_Tout_Tr_Q)
   END_RUNG
   RUNG wire#powerrail
      Contact( "DB1_SalidasExterioresDeMesa".Mesa[#Mesa].Ir_Pos_E1E3 )
      I_Contact( #PosTR_E1 )
   END_RUNG wire#w1
   RUNG wire#powerrail
      Contact( "DB1_SalidasExterioresDeMesa".Mesa[#Mesa].Ir_Pos_E2E4 )
      I_Contact( #PosTR_E2 )
   END_RUNG wire#w1
   // the same network as SCL:
   "FC911_CNT_Tiempo_UHS"(Temporizar := ("DB1_SalidasExterioresDeMesa".Mesa[#Mesa].Ir_Pos_E1E3 AND NOT #PosTR_E1) OR ("DB1_SalidasExterioresDeMesa".Mesa[#Mesa].Ir_Pos_E2E4 AND NOT #PosTR_E2),
                          Valor_Tiempo := #V_TOut_TR,
                          Base_tiempo_ms := 1,
                          Valor_Actual := #TMP_Tout_Tr,
                          Tiempo_OK => #Tmp_Tout_Tr_Q);
END_REGION

REGION Network 29: Marca General Error. "DB900_Estado_Mesas".EstadoVI[numeromesa].Err_TOut_Subida
   RUNG wire#powerrail
      Contact( #EstadoZona.Rearme_CBx )
      S_RS(operand := #EstadoVI.Err_TOut_Subida, s1 := wire#w1)
      S_Coil( #EstadoVI.Error_Mx )
   END_RUNG
   RUNG wire#powerrail
      Contact( #Tmp_Tout_Tr_Q )
      Contact( "DB1_SalidasExterioresDeMesa".Mesa[#Mesa].Ir_Pos_E2E4 )
   END_RUNG wire#w1
   // the same network as SCL:
   IF #EstadoZona.Rearme_CBx THEN
       #EstadoVI.Err_TOut_Subida := FALSE;   // RS flip-flop
   END_IF;
   IF #Tmp_Tout_Tr_Q AND "DB1_SalidasExterioresDeMesa".Mesa[#Mesa].Ir_Pos_E2E4 THEN
       #EstadoVI.Err_TOut_Subida := TRUE;
   END_IF;
   IF #EstadoVI.Err_TOut_Subida THEN #EstadoVI.Error_Mx := TRUE; END_IF;
END_REGION

REGION Network 30: Marca General Error. "DB900_Estado_Mesas".EstadoVI[numeromesa].Err_TOut_Bajada
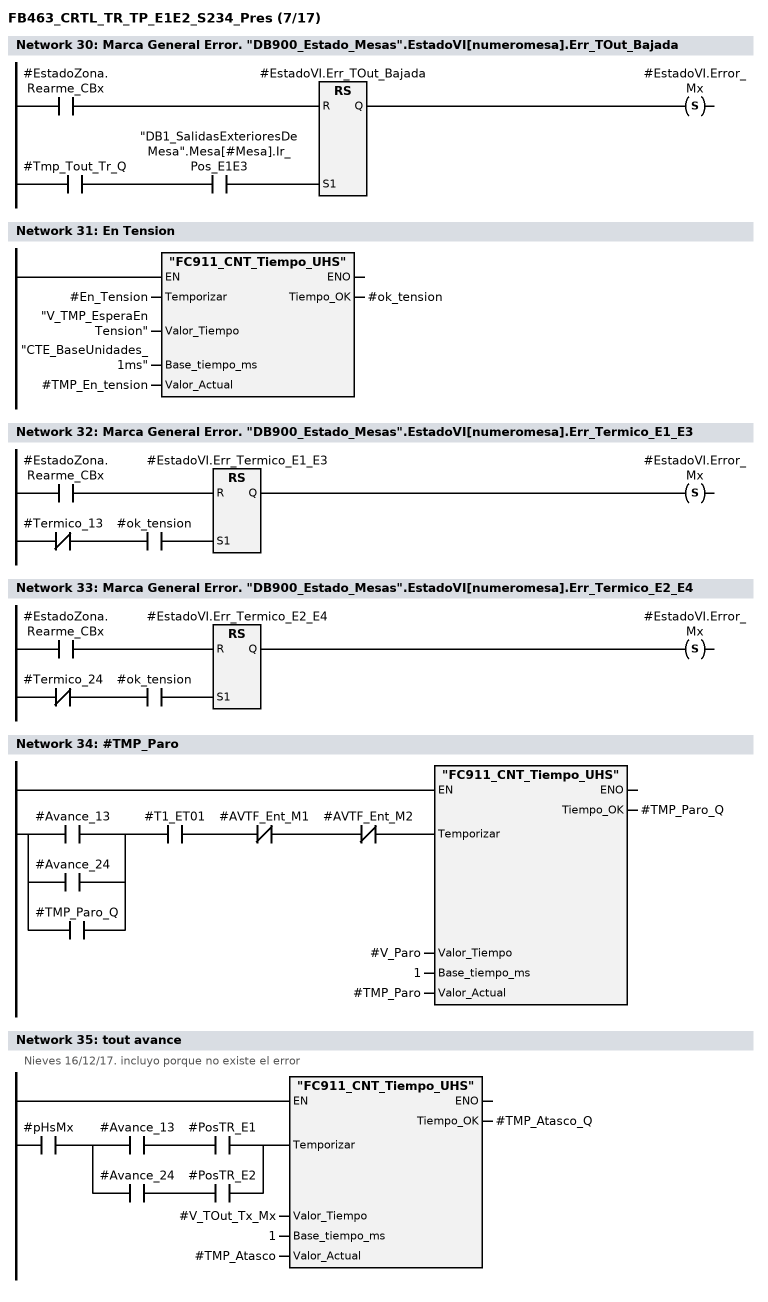
   RUNG wire#powerrail
      Contact( #EstadoZona.Rearme_CBx )
      S_RS(operand := #EstadoVI.Err_TOut_Bajada, s1 := wire#w1)
      S_Coil( #EstadoVI.Error_Mx )
   END_RUNG
   RUNG wire#powerrail
      Contact( #Tmp_Tout_Tr_Q )
      Contact( "DB1_SalidasExterioresDeMesa".Mesa[#Mesa].Ir_Pos_E1E3 )
   END_RUNG wire#w1
   // the same network as SCL:
   IF #EstadoZona.Rearme_CBx THEN
       #EstadoVI.Err_TOut_Bajada := FALSE;   // RS flip-flop
   END_IF;
   IF #Tmp_Tout_Tr_Q AND "DB1_SalidasExterioresDeMesa".Mesa[#Mesa].Ir_Pos_E1E3 THEN
       #EstadoVI.Err_TOut_Bajada := TRUE;
   END_IF;
   IF #EstadoVI.Err_TOut_Bajada THEN #EstadoVI.Error_Mx := TRUE; END_IF;
END_REGION

REGION Network 31: En Tension
   RUNG wire#powerrail
      "FC911_CNT_Tiempo_UHS"(Temporizar := #En_Tension, Valor_Tiempo := "V_TMP_EsperaEnTension", Base_tiempo_ms := "CTE_BaseUnidades_1ms", Valor_Actual := #TMP_En_tension, Tiempo_OK => #ok_tension)
   END_RUNG
   // the same network as SCL:
   "FC911_CNT_Tiempo_UHS"(Temporizar := #En_Tension,
                          Valor_Tiempo := "V_TMP_EsperaEnTension",
                          Base_tiempo_ms := "CTE_BaseUnidades_1ms",
                          Valor_Actual := #TMP_En_tension,
                          Tiempo_OK => #ok_tension);
END_REGION

REGION Network 32: Marca General Error. "DB900_Estado_Mesas".EstadoVI[numeromesa].Err_Termico_E1_E3
   RUNG wire#powerrail
      Contact( #EstadoZona.Rearme_CBx )
      S_RS(operand := #EstadoVI.Err_Termico_E1_E3, s1 := wire#w1)
      S_Coil( #EstadoVI.Error_Mx )
   END_RUNG
   RUNG wire#powerrail
      I_Contact( #Termico_13 )
      Contact( #ok_tension )
   END_RUNG wire#w1
   // the same network as SCL:
   IF #EstadoZona.Rearme_CBx THEN
       #EstadoVI.Err_Termico_E1_E3 := FALSE;   // RS flip-flop
   END_IF;
   IF NOT #Termico_13 AND #ok_tension THEN #EstadoVI.Err_Termico_E1_E3 := TRUE; END_IF;
   IF #EstadoVI.Err_Termico_E1_E3 THEN #EstadoVI.Error_Mx := TRUE; END_IF;
END_REGION

REGION Network 33: Marca General Error. "DB900_Estado_Mesas".EstadoVI[numeromesa].Err_Termico_E2_E4
   RUNG wire#powerrail
      Contact( #EstadoZona.Rearme_CBx )
      S_RS(operand := #EstadoVI.Err_Termico_E2_E4, s1 := wire#w1)
      S_Coil( #EstadoVI.Error_Mx )
   END_RUNG
   RUNG wire#powerrail
      I_Contact( #Termico_24 )
      Contact( #ok_tension )
   END_RUNG wire#w1
   // the same network as SCL:
   IF #EstadoZona.Rearme_CBx THEN
       #EstadoVI.Err_Termico_E2_E4 := FALSE;   // RS flip-flop
   END_IF;
   IF NOT #Termico_24 AND #ok_tension THEN #EstadoVI.Err_Termico_E2_E4 := TRUE; END_IF;
   IF #EstadoVI.Err_Termico_E2_E4 THEN #EstadoVI.Error_Mx := TRUE; END_IF;
END_REGION

REGION Network 34: #TMP_Paro
   RUNG wire#powerrail
      "FC911_CNT_Tiempo_UHS"(Temporizar := wire#w2, Valor_Tiempo := #V_Paro, Base_tiempo_ms := 1, Valor_Actual := #TMP_Paro, Tiempo_OK => #TMP_Paro_Q)
   END_RUNG
   RUNG wire#powerrail
      Contact( #Avance_13 )
      wire#w1
      Contact( #T1_ET01 )
      I_Contact( #AVTF_Ent_M1 )
      I_Contact( #AVTF_Ent_M2 )
   END_RUNG wire#w2
   RUNG wire#powerrail
      Contact( #Avance_24 )
   END_RUNG wire#w1
   RUNG wire#powerrail
      Contact( #TMP_Paro_Q )
   END_RUNG wire#w1
   // the same network as SCL:
   "FC911_CNT_Tiempo_UHS"(Temporizar := (#Avance_13 OR #Avance_24 OR #TMP_Paro_Q) AND #T1_ET01 AND NOT #AVTF_Ent_M1 AND NOT #AVTF_Ent_M2,
                          Valor_Tiempo := #V_Paro,
                          Base_tiempo_ms := 1,
                          Valor_Actual := #TMP_Paro,
                          Tiempo_OK => #TMP_Paro_Q);
END_REGION

REGION Network 35: tout avance
   // Nieves 16/12/17. incluyo porque no existe el error
   RUNG wire#powerrail
      "FC911_CNT_Tiempo_UHS"(Temporizar := wire#w2, Valor_Tiempo := #V_TOut_Tx_Mx, Base_tiempo_ms := 1, Valor_Actual := #TMP_Atasco, Tiempo_OK => #TMP_Atasco_Q)
   END_RUNG
   RUNG wire#powerrail
      Contact( #pHsMx )
      wire#w1
      Contact( #Avance_13 )
      Contact( #PosTR_E1 )
   END_RUNG wire#w2
   RUNG wire#w1
      Contact( #Avance_24 )
      Contact( #PosTR_E2 )
   END_RUNG wire#w2
   // the same network as SCL:
   "FC911_CNT_Tiempo_UHS"(Temporizar := #pHsMx AND ((#Avance_13 AND #PosTR_E1) OR (#Avance_24 AND #PosTR_E2)),
                          Valor_Tiempo := #V_TOut_Tx_Mx,
                          Base_tiempo_ms := 1,
                          Valor_Actual := #TMP_Atasco,
                          Tiempo_OK => #TMP_Atasco_Q);
END_REGION

REGION Network 36: Marca General Error
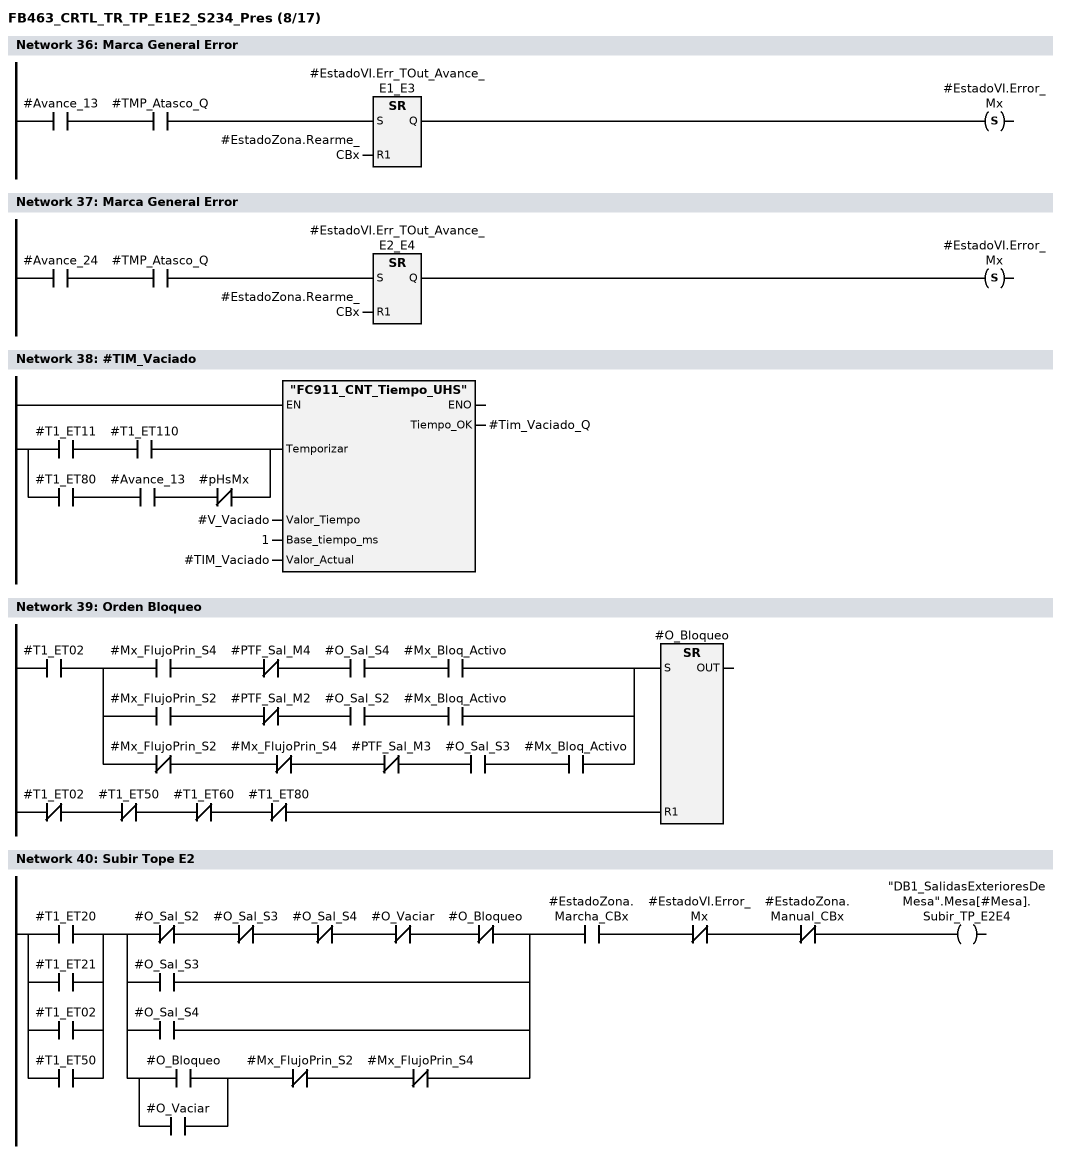
   RUNG wire#powerrail
      Contact( #Avance_13 )
      Contact( #TMP_Atasco_Q )
      S_SR(operand := #EstadoVI.Err_TOut_Avance_E1_E3, r1 := #EstadoZona.Rearme_CBx)
      S_Coil( #EstadoVI.Error_Mx )
   END_RUNG
   // the same network as SCL:
   IF #Avance_13 AND #TMP_Atasco_Q THEN
       #EstadoVI.Err_TOut_Avance_E1_E3 := TRUE;   // SR flip-flop
   END_IF;
   IF #EstadoZona.Rearme_CBx THEN #EstadoVI.Err_TOut_Avance_E1_E3 := FALSE; END_IF;
   IF #EstadoVI.Err_TOut_Avance_E1_E3 THEN #EstadoVI.Error_Mx := TRUE; END_IF;
END_REGION

REGION Network 37: Marca General Error
   RUNG wire#powerrail
      Contact( #Avance_24 )
      Contact( #TMP_Atasco_Q )
      S_SR(operand := #EstadoVI.Err_TOut_Avance_E2_E4, r1 := #EstadoZona.Rearme_CBx)
      S_Coil( #EstadoVI.Error_Mx )
   END_RUNG
   // the same network as SCL:
   IF #Avance_24 AND #TMP_Atasco_Q THEN
       #EstadoVI.Err_TOut_Avance_E2_E4 := TRUE;   // SR flip-flop
   END_IF;
   IF #EstadoZona.Rearme_CBx THEN #EstadoVI.Err_TOut_Avance_E2_E4 := FALSE; END_IF;
   IF #EstadoVI.Err_TOut_Avance_E2_E4 THEN #EstadoVI.Error_Mx := TRUE; END_IF;
END_REGION

REGION Network 38: #TIM_Vaciado
   RUNG wire#powerrail
      "FC911_CNT_Tiempo_UHS"(Temporizar := wire#w1, Valor_Tiempo := #V_Vaciado, Base_tiempo_ms := 1, Valor_Actual := #TIM_Vaciado, Tiempo_OK => #Tim_Vaciado_Q)
   END_RUNG
   RUNG wire#powerrail
      Contact( #T1_ET11 )
      Contact( #T1_ET110 )
   END_RUNG wire#w1
   RUNG wire#powerrail
      Contact( #T1_ET80 )
      Contact( #Avance_13 )
      I_Contact( #pHsMx )
   END_RUNG wire#w1
   // the same network as SCL:
   "FC911_CNT_Tiempo_UHS"(Temporizar := (#T1_ET11 AND #T1_ET110) OR (#T1_ET80 AND #Avance_13 AND NOT #pHsMx),
                          Valor_Tiempo := #V_Vaciado,
                          Base_tiempo_ms := 1,
                          Valor_Actual := #TIM_Vaciado,
                          Tiempo_OK => #Tim_Vaciado_Q);
END_REGION

REGION Network 39: Orden Bloqueo
   RUNG wire#powerrail
      Contact( #T1_ET02 )
      wire#w1
      Contact( #Mx_FlujoPrin_S4 )
      I_Contact( #PTF_Sal_M4 )
      Contact( #O_Sal_S4 )
      Contact( #Mx_Bloq_Activo )
      wire#w2
      S_SR(operand := #O_Bloqueo, r1 := wire#w3)
   END_RUNG
   RUNG wire#w1
      Contact( #Mx_FlujoPrin_S2 )
      I_Contact( #PTF_Sal_M2 )
      Contact( #O_Sal_S2 )
      Contact( #Mx_Bloq_Activo )
   END_RUNG wire#w2
   RUNG wire#w1
      I_Contact( #Mx_FlujoPrin_S2 )
      I_Contact( #Mx_FlujoPrin_S4 )
      I_Contact( #PTF_Sal_M3 )
      Contact( #O_Sal_S3 )
      Contact( #Mx_Bloq_Activo )
   END_RUNG wire#w2
   RUNG wire#powerrail
      I_Contact( #T1_ET02 )
      I_Contact( #T1_ET50 )
      I_Contact( #T1_ET60 )
      I_Contact( #T1_ET80 )
   END_RUNG wire#w3
   // the same network as SCL:
   IF #T1_ET02 AND ((#Mx_FlujoPrin_S4 AND NOT #PTF_Sal_M4 AND #O_Sal_S4 AND #Mx_Bloq_Activo) OR (#Mx_FlujoPrin_S2 AND NOT #PTF_Sal_M2 AND #O_Sal_S2 AND #Mx_Bloq_Activo) OR (NOT #Mx_FlujoPrin_S2 AND NOT #Mx_FlujoPrin_S4 AND NOT #PTF_Sal_M3 AND #O_Sal_S3 AND #Mx_Bloq_Activo)) THEN
       #O_Bloqueo := TRUE;   // SR flip-flop
   END_IF;
   IF NOT #T1_ET02 AND NOT #T1_ET50 AND NOT #T1_ET60 AND NOT #T1_ET80 THEN #O_Bloqueo := FALSE; END_IF;
END_REGION

REGION Network 40: Subir Tope E2
   RUNG wire#powerrail
      Contact( #T1_ET20 )
      wire#w1
      I_Contact( #O_Sal_S2 )
      I_Contact( #O_Sal_S3 )
      I_Contact( #O_Sal_S4 )
      I_Contact( #O_Vaciar )
      I_Contact( #O_Bloqueo )
      wire#w2
      Contact( #EstadoZona.Marcha_CBx )
      I_Contact( #EstadoVI.Error_Mx )
      I_Contact( #EstadoZona.Manual_CBx )
      Coil( "DB1_SalidasExterioresDeMesa".Mesa[#Mesa].Subir_TP_E2E4 )
   END_RUNG
   RUNG wire#powerrail
      Contact( #T1_ET21 )
   END_RUNG wire#w1
   RUNG wire#powerrail
      Contact( #T1_ET02 )
   END_RUNG wire#w1
   RUNG wire#powerrail
      Contact( #T1_ET50 )
   END_RUNG wire#w1
   RUNG wire#w1
      Contact( #O_Sal_S3 )
   END_RUNG wire#w2
   RUNG wire#w1
      Contact( #O_Sal_S4 )
   END_RUNG wire#w2
   RUNG wire#w1
      Contact( #O_Bloqueo )
      wire#w3
      I_Contact( #Mx_FlujoPrin_S2 )
      I_Contact( #Mx_FlujoPrin_S4 )
   END_RUNG wire#w2
   RUNG wire#w1
      Contact( #O_Vaciar )
   END_RUNG wire#w3
   // the same network as SCL:
   "DB1_SalidasExterioresDeMesa".Mesa[#Mesa].Subir_TP_E2E4 := (#T1_ET20 OR #T1_ET21 OR #T1_ET02 OR #T1_ET50) AND ((NOT #O_Sal_S2 AND NOT #O_Sal_S3 AND NOT #O_Sal_S4 AND NOT #O_Vaciar AND NOT #O_Bloqueo) OR #O_Sal_S3 OR #O_Sal_S4 OR ((#O_Bloqueo OR #O_Vaciar) AND NOT #Mx_FlujoPrin_S2 AND NOT #Mx_FlujoPrin_S4)) AND #EstadoZona.Marcha_CBx AND NOT #EstadoVI.Error_Mx AND NOT #EstadoZona.Manual_CBx;
END_REGION

REGION Network 41: Subir Tope E2
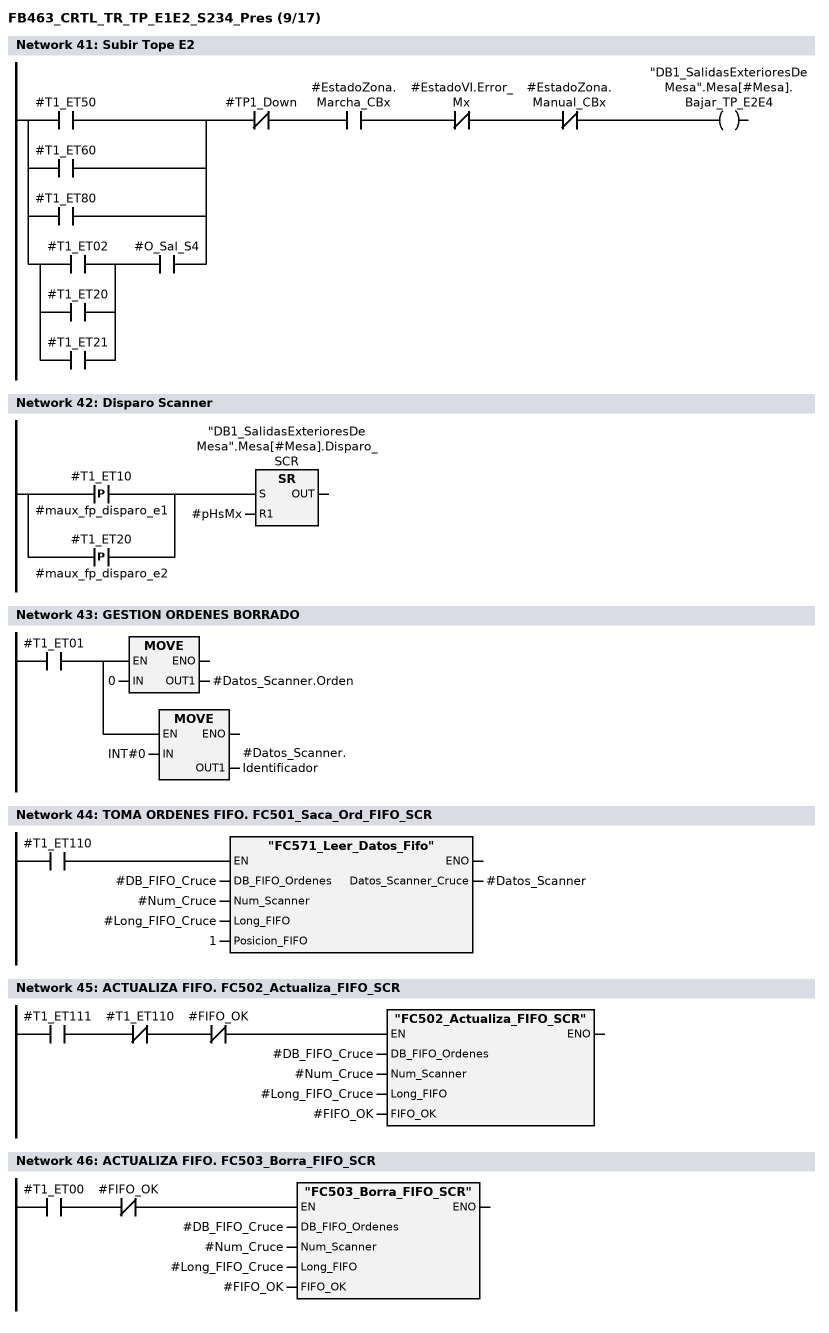
   RUNG wire#powerrail
      Contact( #T1_ET50 )
      wire#w1
      I_Contact( #TP1_Down )
      Contact( #EstadoZona.Marcha_CBx )
      I_Contact( #EstadoVI.Error_Mx )
      I_Contact( #EstadoZona.Manual_CBx )
      Coil( "DB1_SalidasExterioresDeMesa".Mesa[#Mesa].Bajar_TP_E2E4 )
   END_RUNG
   RUNG wire#powerrail
      Contact( #T1_ET60 )
   END_RUNG wire#w1
   RUNG wire#powerrail
      Contact( #T1_ET80 )
   END_RUNG wire#w1
   RUNG wire#powerrail
      Contact( #T1_ET02 )
      wire#w2
      Contact( #O_Sal_S4 )
   END_RUNG wire#w1
   RUNG wire#powerrail
      Contact( #T1_ET20 )
   END_RUNG wire#w2
   RUNG wire#powerrail
      Contact( #T1_ET21 )
   END_RUNG wire#w2
   // the same network as SCL:
   "DB1_SalidasExterioresDeMesa".Mesa[#Mesa].Bajar_TP_E2E4 := (#T1_ET50 OR #T1_ET60 OR #T1_ET80 OR ((#T1_ET02 OR #T1_ET20 OR #T1_ET21) AND #O_Sal_S4)) AND NOT #TP1_Down AND #EstadoZona.Marcha_CBx AND NOT #EstadoVI.Error_Mx AND NOT #EstadoZona.Manual_CBx;
END_REGION

REGION Network 42: Disparo Scanner
   RUNG wire#powerrail
      P_Contact(operand := #T1_ET10, bit := #maux_fp_disparo_e1)
      wire#w1
      S_SR(operand := "DB1_SalidasExterioresDeMesa".Mesa[#Mesa].Disparo_SCR, r1 := #pHsMx)
   END_RUNG
   RUNG wire#powerrail
      P_Contact(operand := #T1_ET20, bit := #maux_fp_disparo_e2)
   END_RUNG wire#w1
   // the same network as SCL:
   #_w1 := #T1_ET10 AND NOT #maux_fp_disparo_e1;   // rising edge of #T1_ET10
   #maux_fp_disparo_e1 := #T1_ET10;
   #_w2 := #T1_ET20 AND NOT #maux_fp_disparo_e2;   // rising edge of #T1_ET20
   #maux_fp_disparo_e2 := #T1_ET20;
   IF #_w1 OR #_w2 THEN
       "DB1_SalidasExterioresDeMesa".Mesa[#Mesa].Disparo_SCR := TRUE;   // SR flip-flop
   END_IF;
   IF #pHsMx THEN "DB1_SalidasExterioresDeMesa".Mesa[#Mesa].Disparo_SCR := FALSE; END_IF;
END_REGION

REGION Network 43: GESTION ORDENES BORRADO
   RUNG wire#powerrail
      Contact( #T1_ET01 )
      wire#w1
      { S7_GenerateENO := "TRUE" } Move(in := 0, out1 => #Datos_Scanner.Orden)
   END_RUNG
   RUNG wire#w1
      { S7_GenerateENO := "TRUE" } Move(in := INT#0, out1 => #Datos_Scanner.Identificador)
   END_RUNG
   // the same network as SCL:
   IF #T1_ET01 THEN
       #Datos_Scanner.Orden := 0;
       #Datos_Scanner.Identificador := INT#0;
   END_IF;
END_REGION

REGION Network 44: TOMA ORDENES FIFO. FC501_Saca_Ord_FIFO_SCR
   RUNG wire#powerrail
      Contact( #T1_ET110 )
      "FC571_Leer_Datos_Fifo"(DB_FIFO_Ordenes := #DB_FIFO_Cruce, Num_Scanner := #Num_Cruce, Long_FIFO := #Long_FIFO_Cruce, Posicion_FIFO := 1, Datos_Scanner_Cruce => #Datos_Scanner)
   END_RUNG
   // the same network as SCL:
   IF #T1_ET110 THEN
       "FC571_Leer_Datos_Fifo"(DB_FIFO_Ordenes := #DB_FIFO_Cruce,
                               Num_Scanner := #Num_Cruce,
                               Long_FIFO := #Long_FIFO_Cruce,
                               Posicion_FIFO := 1,
                               Datos_Scanner_Cruce => #Datos_Scanner);
   END_IF;
END_REGION

REGION Network 45: ACTUALIZA FIFO. FC502_Actualiza_FIFO_SCR
   RUNG wire#powerrail
      Contact( #T1_ET111 )
      I_Contact( #T1_ET110 )
      I_Contact( #FIFO_OK )
      "FC502_Actualiza_FIFO_SCR"(DB_FIFO_Ordenes := #DB_FIFO_Cruce, Num_Scanner := #Num_Cruce, Long_FIFO := #Long_FIFO_Cruce, FIFO_OK := #FIFO_OK)
   END_RUNG
   // the same network as SCL:
   IF #T1_ET111 AND NOT #T1_ET110 AND NOT #FIFO_OK THEN
       "FC502_Actualiza_FIFO_SCR"(DB_FIFO_Ordenes := #DB_FIFO_Cruce,
                               Num_Scanner := #Num_Cruce,
                               Long_FIFO := #Long_FIFO_Cruce,
                               FIFO_OK := #FIFO_OK);
   END_IF;
END_REGION

REGION Network 46: ACTUALIZA FIFO. FC503_Borra_FIFO_SCR
   RUNG wire#powerrail
      Contact( #T1_ET00 )
      I_Contact( #FIFO_OK )
      "FC503_Borra_FIFO_SCR"(DB_FIFO_Ordenes := #DB_FIFO_Cruce, Num_Scanner := #Num_Cruce, Long_FIFO := #Long_FIFO_Cruce, FIFO_OK := #FIFO_OK)
   END_RUNG
   // the same network as SCL:
   IF #T1_ET00 AND NOT #FIFO_OK THEN
       "FC503_Borra_FIFO_SCR"(DB_FIFO_Ordenes := #DB_FIFO_Cruce,
                              Num_Scanner := #Num_Cruce,
                              Long_FIFO := #Long_FIFO_Cruce,
                              FIFO_OK := #FIFO_OK);
   END_IF;
END_REGION

REGION Network 47: "FC506_PASAR_ORD_SCR". S3
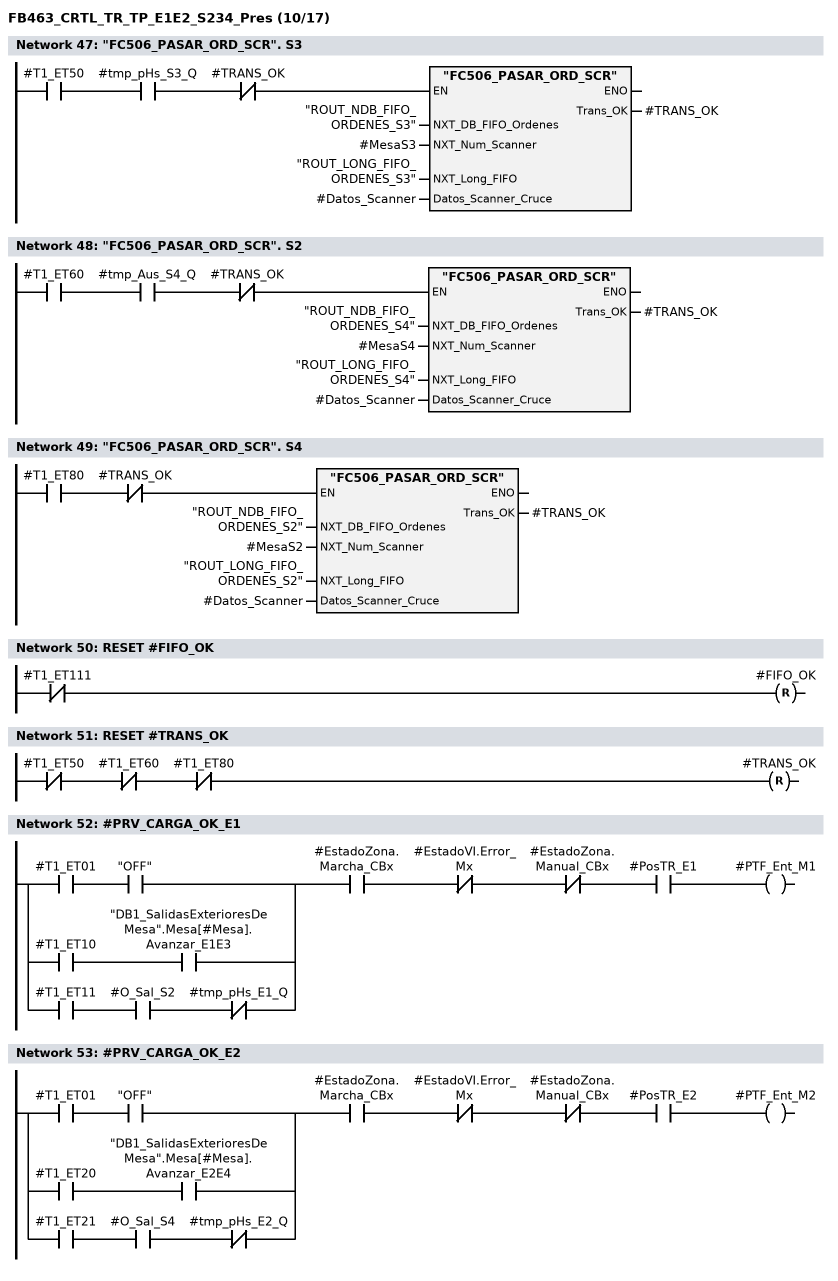
   RUNG wire#powerrail
      Contact( #T1_ET50 )
      Contact( #tmp_pHs_S3_Q )
      I_Contact( #TRANS_OK )
      "FC506_PASAR_ORD_SCR"(NXT_DB_FIFO_Ordenes := "ROUT_NDB_FIFO_ORDENES_S3", NXT_Num_Scanner := #MesaS3, NXT_Long_FIFO := "ROUT_LONG_FIFO_ORDENES_S3", Datos_Scanner_Cruce := #Datos_Scanner, Trans_OK => #TRANS_OK)
   END_RUNG
   // the same network as SCL:
   IF #T1_ET50 AND #tmp_pHs_S3_Q AND NOT #TRANS_OK THEN
       "FC506_PASAR_ORD_SCR"(NXT_DB_FIFO_Ordenes := "ROUT_NDB_FIFO_ORDENES_S3",
                             NXT_Num_Scanner := #MesaS3,
                             NXT_Long_FIFO := "ROUT_LONG_FIFO_ORDENES_S3",
                             Datos_Scanner_Cruce := #Datos_Scanner,
                             Trans_OK => #TRANS_OK);
   END_IF;
END_REGION

REGION Network 48: "FC506_PASAR_ORD_SCR". S2
   RUNG wire#powerrail
      Contact( #T1_ET60 )
      Contact( #tmp_Aus_S4_Q )
      I_Contact( #TRANS_OK )
      "FC506_PASAR_ORD_SCR"(NXT_DB_FIFO_Ordenes := "ROUT_NDB_FIFO_ORDENES_S4", NXT_Num_Scanner := #MesaS4, NXT_Long_FIFO := "ROUT_LONG_FIFO_ORDENES_S4", Datos_Scanner_Cruce := #Datos_Scanner, Trans_OK => #TRANS_OK)
   END_RUNG
   // the same network as SCL:
   IF #T1_ET60 AND #tmp_Aus_S4_Q AND NOT #TRANS_OK THEN
       "FC506_PASAR_ORD_SCR"(NXT_DB_FIFO_Ordenes := "ROUT_NDB_FIFO_ORDENES_S4",
                             NXT_Num_Scanner := #MesaS4,
                             NXT_Long_FIFO := "ROUT_LONG_FIFO_ORDENES_S4",
                             Datos_Scanner_Cruce := #Datos_Scanner,
                             Trans_OK => #TRANS_OK);
   END_IF;
END_REGION

REGION Network 49: "FC506_PASAR_ORD_SCR". S4
   RUNG wire#powerrail
      Contact( #T1_ET80 )
      I_Contact( #TRANS_OK )
      "FC506_PASAR_ORD_SCR"(NXT_DB_FIFO_Ordenes := "ROUT_NDB_FIFO_ORDENES_S2", NXT_Num_Scanner := #MesaS2, NXT_Long_FIFO := "ROUT_LONG_FIFO_ORDENES_S2", Datos_Scanner_Cruce := #Datos_Scanner, Trans_OK => #TRANS_OK)
   END_RUNG
   // the same network as SCL:
   IF #T1_ET80 AND NOT #TRANS_OK THEN
       "FC506_PASAR_ORD_SCR"(NXT_DB_FIFO_Ordenes := "ROUT_NDB_FIFO_ORDENES_S2",
                             NXT_Num_Scanner := #MesaS2,
                             NXT_Long_FIFO := "ROUT_LONG_FIFO_ORDENES_S2",
                             Datos_Scanner_Cruce := #Datos_Scanner,
                             Trans_OK => #TRANS_OK);
   END_IF;
END_REGION

REGION Network 50: RESET #FIFO_OK
   RUNG wire#powerrail
      I_Contact( #T1_ET111 )
      R_Coil( #FIFO_OK )
   END_RUNG
   // the same network as SCL:
   IF NOT #T1_ET111 THEN #FIFO_OK := FALSE; END_IF;
END_REGION

REGION Network 51: RESET #TRANS_OK
   RUNG wire#powerrail
      I_Contact( #T1_ET50 )
      I_Contact( #T1_ET60 )
      I_Contact( #T1_ET80 )
      R_Coil( #TRANS_OK )
   END_RUNG
   // the same network as SCL:
   IF NOT #T1_ET50 AND NOT #T1_ET60 AND NOT #T1_ET80 THEN #TRANS_OK := FALSE; END_IF;
END_REGION

REGION Network 52: #PRV_CARGA_OK_E1
   RUNG wire#powerrail
      Contact( #T1_ET01 )
      Contact( "OFF" )
      wire#w1
      Contact( #EstadoZona.Marcha_CBx )
      I_Contact( #EstadoVI.Error_Mx )
      I_Contact( #EstadoZona.Manual_CBx )
      Contact( #PosTR_E1 )
      Coil( #PTF_Ent_M1 )
   END_RUNG
   RUNG wire#powerrail
      Contact( #T1_ET10 )
      Contact( "DB1_SalidasExterioresDeMesa".Mesa[#Mesa].Avanzar_E1E3 )
   END_RUNG wire#w1
   RUNG wire#powerrail
      Contact( #T1_ET11 )
      Contact( #O_Sal_S2 )
      I_Contact( #tmp_pHs_E1_Q )
   END_RUNG wire#w1
   // the same network as SCL:
   #PTF_Ent_M1 := ((#T1_ET01 AND "OFF") OR (#T1_ET10 AND "DB1_SalidasExterioresDeMesa".Mesa[#Mesa].Avanzar_E1E3) OR (#T1_ET11 AND #O_Sal_S2 AND NOT #tmp_pHs_E1_Q)) AND #EstadoZona.Marcha_CBx AND NOT #EstadoVI.Error_Mx AND NOT #EstadoZona.Manual_CBx AND #PosTR_E1;
END_REGION

REGION Network 53: #PRV_CARGA_OK_E2
   RUNG wire#powerrail
      Contact( #T1_ET01 )
      Contact( "OFF" )
      wire#w1
      Contact( #EstadoZona.Marcha_CBx )
      I_Contact( #EstadoVI.Error_Mx )
      I_Contact( #EstadoZona.Manual_CBx )
      Contact( #PosTR_E2 )
      Coil( #PTF_Ent_M2 )
   END_RUNG
   RUNG wire#powerrail
      Contact( #T1_ET20 )
      Contact( "DB1_SalidasExterioresDeMesa".Mesa[#Mesa].Avanzar_E2E4 )
   END_RUNG wire#w1
   RUNG wire#powerrail
      Contact( #T1_ET21 )
      Contact( #O_Sal_S4 )
      I_Contact( #tmp_pHs_E2_Q )
   END_RUNG wire#w1
   // the same network as SCL:
   #PTF_Ent_M2 := ((#T1_ET01 AND "OFF") OR (#T1_ET20 AND "DB1_SalidasExterioresDeMesa".Mesa[#Mesa].Avanzar_E2E4) OR (#T1_ET21 AND #O_Sal_S4 AND NOT #tmp_pHs_E2_Q)) AND #EstadoZona.Marcha_CBx AND NOT #EstadoVI.Error_Mx AND NOT #EstadoZona.Manual_CBx AND #PosTR_E2;
END_REGION

REGION Network 54: #NXT_AVTF_S2
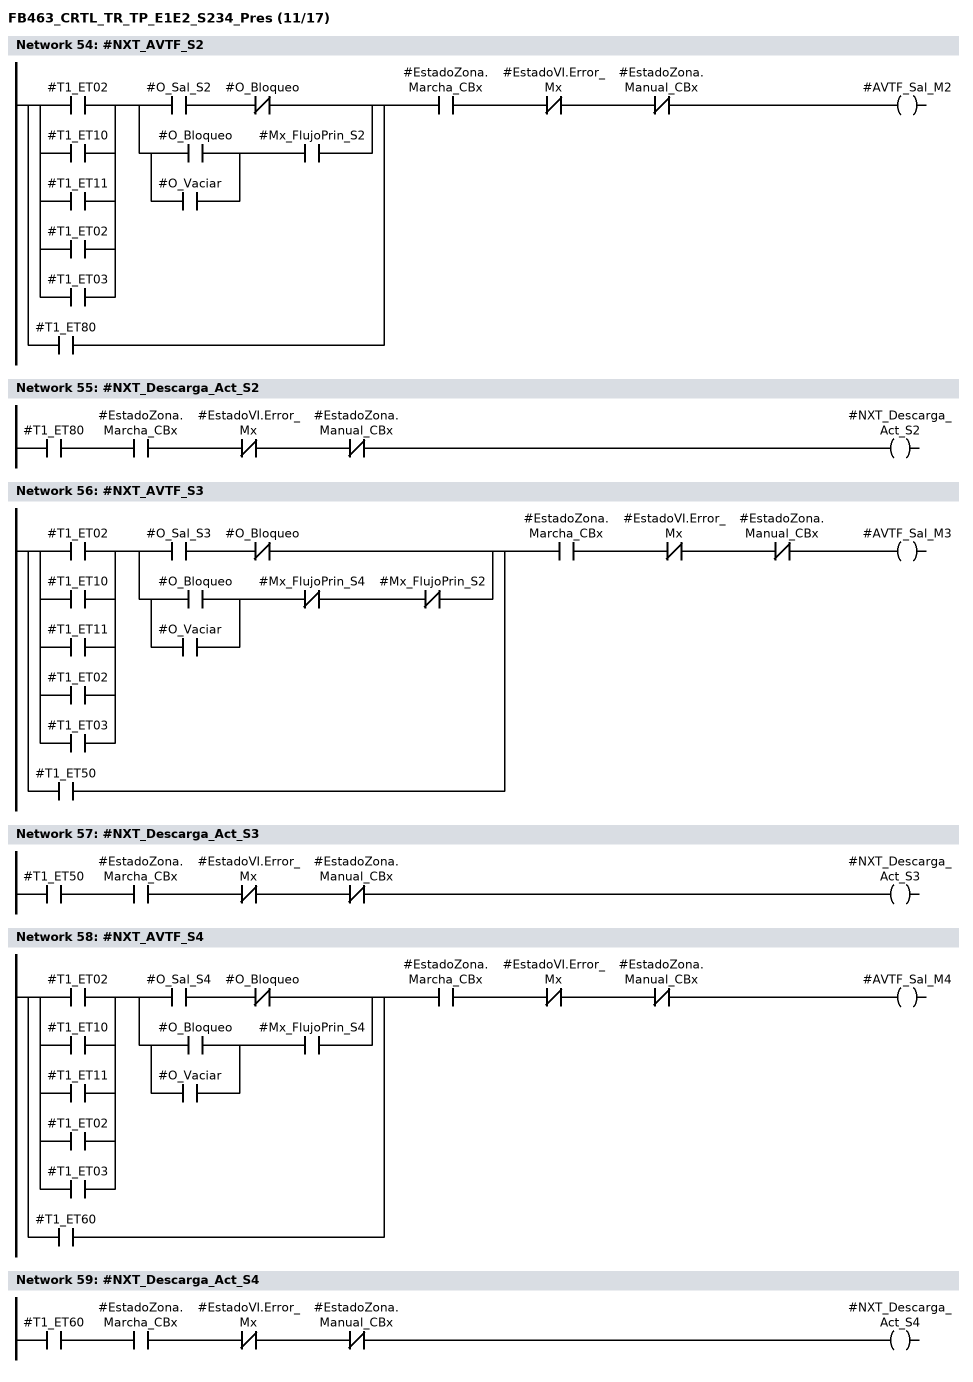
   RUNG wire#powerrail
      Contact( #T1_ET02 )
      wire#w1
      Contact( #O_Sal_S2 )
      I_Contact( #O_Bloqueo )
      wire#w2
      Contact( #EstadoZona.Marcha_CBx )
      I_Contact( #EstadoVI.Error_Mx )
      I_Contact( #EstadoZona.Manual_CBx )
      Coil( #AVTF_Sal_M2 )
   END_RUNG
   RUNG wire#powerrail
      Contact( #T1_ET10 )
   END_RUNG wire#w1
   RUNG wire#powerrail
      Contact( #T1_ET11 )
   END_RUNG wire#w1
   RUNG wire#powerrail
      Contact( #T1_ET02 )
   END_RUNG wire#w1
   RUNG wire#powerrail
      Contact( #T1_ET03 )
   END_RUNG wire#w1
   RUNG wire#w1
      Contact( #O_Bloqueo )
      wire#w3
      Contact( #Mx_FlujoPrin_S2 )
   END_RUNG wire#w2
   RUNG wire#w1
      Contact( #O_Vaciar )
   END_RUNG wire#w3
   RUNG wire#powerrail
      Contact( #T1_ET80 )
   END_RUNG wire#w2
   // the same network as SCL:
   #AVTF_Sal_M2 := (((#T1_ET02 OR #T1_ET10 OR #T1_ET11 OR #T1_ET02 OR #T1_ET03) AND ((#O_Sal_S2 AND NOT #O_Bloqueo) OR ((#O_Bloqueo OR #O_Vaciar) AND #Mx_FlujoPrin_S2))) OR #T1_ET80) AND #EstadoZona.Marcha_CBx AND NOT #EstadoVI.Error_Mx AND NOT #EstadoZona.Manual_CBx;
END_REGION

REGION Network 55: #NXT_Descarga_Act_S2
   RUNG wire#powerrail
      Contact( #T1_ET80 )
      Contact( #EstadoZona.Marcha_CBx )
      I_Contact( #EstadoVI.Error_Mx )
      I_Contact( #EstadoZona.Manual_CBx )
      Coil( #NXT_Descarga_Act_S2 )
   END_RUNG
   // the same network as SCL:
   #NXT_Descarga_Act_S2 := #T1_ET80 AND #EstadoZona.Marcha_CBx AND NOT #EstadoVI.Error_Mx AND NOT #EstadoZona.Manual_CBx;
END_REGION

REGION Network 56: #NXT_AVTF_S3
   RUNG wire#powerrail
      Contact( #T1_ET02 )
      wire#w1
      Contact( #O_Sal_S3 )
      I_Contact( #O_Bloqueo )
      wire#w2
      Contact( #EstadoZona.Marcha_CBx )
      I_Contact( #EstadoVI.Error_Mx )
      I_Contact( #EstadoZona.Manual_CBx )
      Coil( #AVTF_Sal_M3 )
   END_RUNG
   RUNG wire#powerrail
      Contact( #T1_ET10 )
   END_RUNG wire#w1
   RUNG wire#powerrail
      Contact( #T1_ET11 )
   END_RUNG wire#w1
   RUNG wire#powerrail
      Contact( #T1_ET02 )
   END_RUNG wire#w1
   RUNG wire#powerrail
      Contact( #T1_ET03 )
   END_RUNG wire#w1
   RUNG wire#w1
      Contact( #O_Bloqueo )
      wire#w3
      I_Contact( #Mx_FlujoPrin_S4 )
      I_Contact( #Mx_FlujoPrin_S2 )
   END_RUNG wire#w2
   RUNG wire#w1
      Contact( #O_Vaciar )
   END_RUNG wire#w3
   RUNG wire#powerrail
      Contact( #T1_ET50 )
   END_RUNG wire#w2
   // the same network as SCL:
   #AVTF_Sal_M3 := (((#T1_ET02 OR #T1_ET10 OR #T1_ET11 OR #T1_ET02 OR #T1_ET03) AND ((#O_Sal_S3 AND NOT #O_Bloqueo) OR ((#O_Bloqueo OR #O_Vaciar) AND NOT #Mx_FlujoPrin_S4 AND NOT #Mx_FlujoPrin_S2))) OR #T1_ET50) AND #EstadoZona.Marcha_CBx AND NOT #EstadoVI.Error_Mx AND NOT #EstadoZona.Manual_CBx;
END_REGION

REGION Network 57: #NXT_Descarga_Act_S3
   RUNG wire#powerrail
      Contact( #T1_ET50 )
      Contact( #EstadoZona.Marcha_CBx )
      I_Contact( #EstadoVI.Error_Mx )
      I_Contact( #EstadoZona.Manual_CBx )
      Coil( #NXT_Descarga_Act_S3 )
   END_RUNG
   // the same network as SCL:
   #NXT_Descarga_Act_S3 := #T1_ET50 AND #EstadoZona.Marcha_CBx AND NOT #EstadoVI.Error_Mx AND NOT #EstadoZona.Manual_CBx;
END_REGION

REGION Network 58: #NXT_AVTF_S4
   RUNG wire#powerrail
      Contact( #T1_ET02 )
      wire#w1
      Contact( #O_Sal_S4 )
      I_Contact( #O_Bloqueo )
      wire#w2
      Contact( #EstadoZona.Marcha_CBx )
      I_Contact( #EstadoVI.Error_Mx )
      I_Contact( #EstadoZona.Manual_CBx )
      Coil( #AVTF_Sal_M4 )
   END_RUNG
   RUNG wire#powerrail
      Contact( #T1_ET10 )
   END_RUNG wire#w1
   RUNG wire#powerrail
      Contact( #T1_ET11 )
   END_RUNG wire#w1
   RUNG wire#powerrail
      Contact( #T1_ET02 )
   END_RUNG wire#w1
   RUNG wire#powerrail
      Contact( #T1_ET03 )
   END_RUNG wire#w1
   RUNG wire#w1
      Contact( #O_Bloqueo )
      wire#w3
      Contact( #Mx_FlujoPrin_S4 )
   END_RUNG wire#w2
   RUNG wire#w1
      Contact( #O_Vaciar )
   END_RUNG wire#w3
   RUNG wire#powerrail
      Contact( #T1_ET60 )
   END_RUNG wire#w2
   // the same network as SCL:
   #AVTF_Sal_M4 := (((#T1_ET02 OR #T1_ET10 OR #T1_ET11 OR #T1_ET02 OR #T1_ET03) AND ((#O_Sal_S4 AND NOT #O_Bloqueo) OR ((#O_Bloqueo OR #O_Vaciar) AND #Mx_FlujoPrin_S4))) OR #T1_ET60) AND #EstadoZona.Marcha_CBx AND NOT #EstadoVI.Error_Mx AND NOT #EstadoZona.Manual_CBx;
END_REGION

REGION Network 59: #NXT_Descarga_Act_S4
   RUNG wire#powerrail
      Contact( #T1_ET60 )
      Contact( #EstadoZona.Marcha_CBx )
      I_Contact( #EstadoVI.Error_Mx )
      I_Contact( #EstadoZona.Manual_CBx )
      Coil( #NXT_Descarga_Act_S4 )
   END_RUNG
   // the same network as SCL:
   #NXT_Descarga_Act_S4 := #T1_ET60 AND #EstadoZona.Marcha_CBx AND NOT #EstadoVI.Error_Mx AND NOT #EstadoZona.Manual_CBx;
END_REGION

REGION Network 60: Subir Tope E1
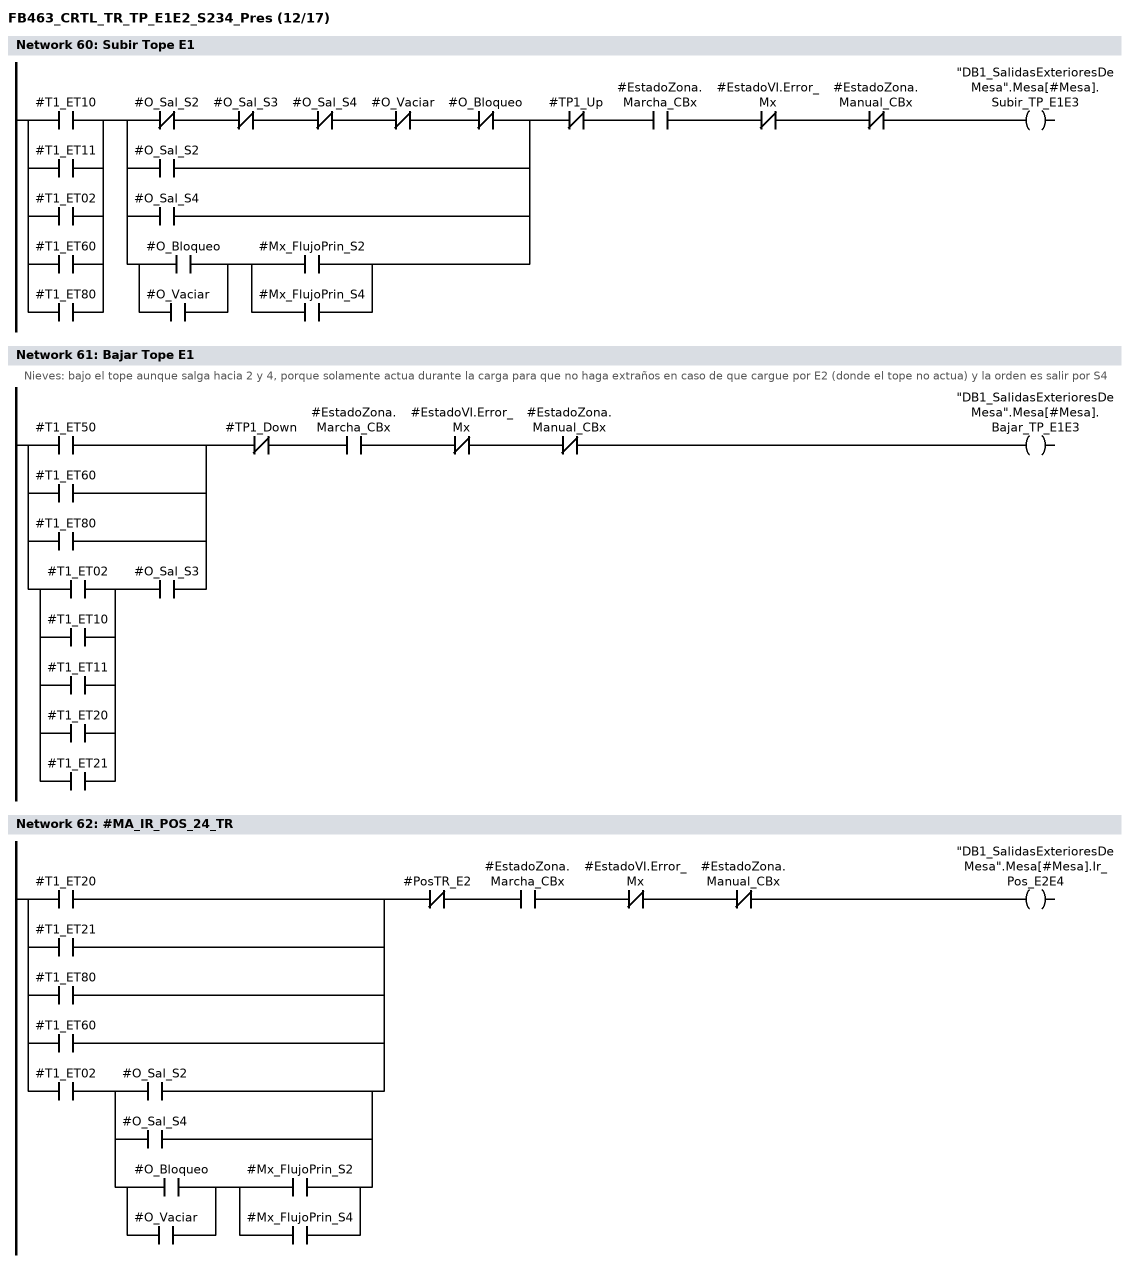
   RUNG wire#powerrail
      Contact( #T1_ET10 )
      wire#w1
      I_Contact( #O_Sal_S2 )
      I_Contact( #O_Sal_S3 )
      I_Contact( #O_Sal_S4 )
      I_Contact( #O_Vaciar )
      I_Contact( #O_Bloqueo )
      wire#w2
      I_Contact( #TP1_Up )
      Contact( #EstadoZona.Marcha_CBx )
      I_Contact( #EstadoVI.Error_Mx )
      I_Contact( #EstadoZona.Manual_CBx )
      Coil( "DB1_SalidasExterioresDeMesa".Mesa[#Mesa].Subir_TP_E1E3 )
   END_RUNG
   RUNG wire#powerrail
      Contact( #T1_ET11 )
   END_RUNG wire#w1
   RUNG wire#powerrail
      Contact( #T1_ET02 )
   END_RUNG wire#w1
   RUNG wire#powerrail
      Contact( #T1_ET60 )
   END_RUNG wire#w1
   RUNG wire#powerrail
      Contact( #T1_ET80 )
   END_RUNG wire#w1
   RUNG wire#w1
      Contact( #O_Sal_S2 )
   END_RUNG wire#w2
   RUNG wire#w1
      Contact( #O_Sal_S4 )
   END_RUNG wire#w2
   RUNG wire#w1
      Contact( #O_Bloqueo )
      wire#w3
      Contact( #Mx_FlujoPrin_S2 )
   END_RUNG wire#w2
   RUNG wire#w1
      Contact( #O_Vaciar )
   END_RUNG wire#w3
   RUNG wire#w3
      Contact( #Mx_FlujoPrin_S4 )
   END_RUNG wire#w2
   // the same network as SCL:
   "DB1_SalidasExterioresDeMesa".Mesa[#Mesa].Subir_TP_E1E3 := (#T1_ET10 OR #T1_ET11 OR #T1_ET02 OR #T1_ET60 OR #T1_ET80) AND ((NOT #O_Sal_S2 AND NOT #O_Sal_S3 AND NOT #O_Sal_S4 AND NOT #O_Vaciar AND NOT #O_Bloqueo) OR #O_Sal_S2 OR #O_Sal_S4 OR ((#O_Bloqueo OR #O_Vaciar) AND (#Mx_FlujoPrin_S2 OR #Mx_FlujoPrin_S4))) AND NOT #TP1_Up AND #EstadoZona.Marcha_CBx AND NOT #EstadoVI.Error_Mx AND NOT #EstadoZona.Manual_CBx;
END_REGION

REGION Network 61: Bajar Tope E1
   // Nieves: bajo el tope aunque salga hacia 2 y 4, porque solamente actua durante la carga para que no haga extraños en caso de que cargue por E2 (donde el tope no actua) y la orden es salir por S4
   RUNG wire#powerrail
      Contact( #T1_ET50 )
      wire#w1
      I_Contact( #TP1_Down )
      Contact( #EstadoZona.Marcha_CBx )
      I_Contact( #EstadoVI.Error_Mx )
      I_Contact( #EstadoZona.Manual_CBx )
      Coil( "DB1_SalidasExterioresDeMesa".Mesa[#Mesa].Bajar_TP_E1E3 )
   END_RUNG
   RUNG wire#powerrail
      Contact( #T1_ET60 )
   END_RUNG wire#w1
   RUNG wire#powerrail
      Contact( #T1_ET80 )
   END_RUNG wire#w1
   RUNG wire#powerrail
      Contact( #T1_ET02 )
      wire#w2
      Contact( #O_Sal_S3 )
   END_RUNG wire#w1
   RUNG wire#powerrail
      Contact( #T1_ET10 )
   END_RUNG wire#w2
   RUNG wire#powerrail
      Contact( #T1_ET11 )
   END_RUNG wire#w2
   RUNG wire#powerrail
      Contact( #T1_ET20 )
   END_RUNG wire#w2
   RUNG wire#powerrail
      Contact( #T1_ET21 )
   END_RUNG wire#w2
   // the same network as SCL:
   "DB1_SalidasExterioresDeMesa".Mesa[#Mesa].Bajar_TP_E1E3 := (#T1_ET50 OR #T1_ET60 OR #T1_ET80 OR ((#T1_ET02 OR #T1_ET10 OR #T1_ET11 OR #T1_ET20 OR #T1_ET21) AND #O_Sal_S3)) AND NOT #TP1_Down AND #EstadoZona.Marcha_CBx AND NOT #EstadoVI.Error_Mx AND NOT #EstadoZona.Manual_CBx;
END_REGION

REGION Network 62: #MA_IR_POS_24_TR
   RUNG wire#powerrail
      Contact( #T1_ET20 )
      wire#w1
      I_Contact( #PosTR_E2 )
      Contact( #EstadoZona.Marcha_CBx )
      I_Contact( #EstadoVI.Error_Mx )
      I_Contact( #EstadoZona.Manual_CBx )
      Coil( "DB1_SalidasExterioresDeMesa".Mesa[#Mesa].Ir_Pos_E2E4 )
   END_RUNG
   RUNG wire#powerrail
      Contact( #T1_ET21 )
   END_RUNG wire#w1
   RUNG wire#powerrail
      Contact( #T1_ET80 )
   END_RUNG wire#w1
   RUNG wire#powerrail
      Contact( #T1_ET60 )
   END_RUNG wire#w1
   RUNG wire#powerrail
      Contact( #T1_ET02 )
      wire#w2
      Contact( #O_Sal_S2 )
   END_RUNG wire#w1
   RUNG wire#w2
      Contact( #O_Sal_S4 )
   END_RUNG wire#w1
   RUNG wire#w2
      Contact( #O_Bloqueo )
      wire#w3
      Contact( #Mx_FlujoPrin_S2 )
   END_RUNG wire#w1
   RUNG wire#w2
      Contact( #O_Vaciar )
   END_RUNG wire#w3
   RUNG wire#w3
      Contact( #Mx_FlujoPrin_S4 )
   END_RUNG wire#w1
   // the same network as SCL:
   "DB1_SalidasExterioresDeMesa".Mesa[#Mesa].Ir_Pos_E2E4 := (#T1_ET20 OR #T1_ET21 OR #T1_ET80 OR #T1_ET60 OR (#T1_ET02 AND (#O_Sal_S2 OR #O_Sal_S4 OR ((#O_Bloqueo OR #O_Vaciar) AND (#Mx_FlujoPrin_S2 OR #Mx_FlujoPrin_S4))))) AND NOT #PosTR_E2 AND #EstadoZona.Marcha_CBx AND NOT #EstadoVI.Error_Mx AND NOT #EstadoZona.Manual_CBx;
END_REGION

REGION Network 63: #MA_IR_POS_13_T
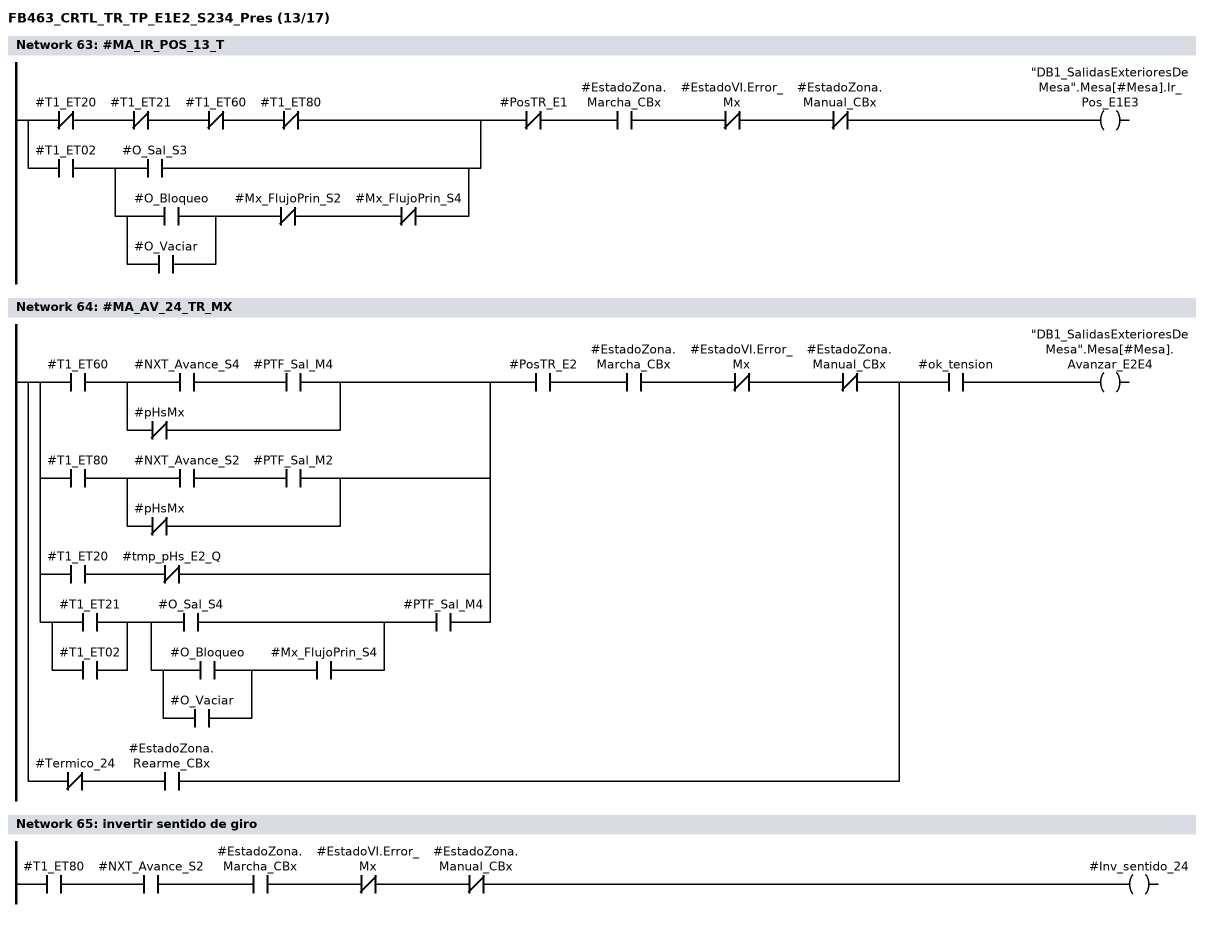
   RUNG wire#powerrail
      I_Contact( #T1_ET20 )
      I_Contact( #T1_ET21 )
      I_Contact( #T1_ET60 )
      I_Contact( #T1_ET80 )
      wire#w1
      I_Contact( #PosTR_E1 )
      Contact( #EstadoZona.Marcha_CBx )
      I_Contact( #EstadoVI.Error_Mx )
      I_Contact( #EstadoZona.Manual_CBx )
      Coil( "DB1_SalidasExterioresDeMesa".Mesa[#Mesa].Ir_Pos_E1E3 )
   END_RUNG
   RUNG wire#powerrail
      Contact( #T1_ET02 )
      wire#w2
      Contact( #O_Sal_S3 )
   END_RUNG wire#w1
   RUNG wire#w2
      Contact( #O_Bloqueo )
      wire#w3
      I_Contact( #Mx_FlujoPrin_S2 )
      I_Contact( #Mx_FlujoPrin_S4 )
   END_RUNG wire#w1
   RUNG wire#w2
      Contact( #O_Vaciar )
   END_RUNG wire#w3
   // the same network as SCL:
   "DB1_SalidasExterioresDeMesa".Mesa[#Mesa].Ir_Pos_E1E3 := ((NOT #T1_ET20 AND NOT #T1_ET21 AND NOT #T1_ET60 AND NOT #T1_ET80) OR (#T1_ET02 AND (#O_Sal_S3 OR ((#O_Bloqueo OR #O_Vaciar) AND NOT #Mx_FlujoPrin_S2 AND NOT #Mx_FlujoPrin_S4)))) AND NOT #PosTR_E1 AND #EstadoZona.Marcha_CBx AND NOT #EstadoVI.Error_Mx AND NOT #EstadoZona.Manual_CBx;
END_REGION

REGION Network 64: #MA_AV_24_TR_MX
   RUNG wire#powerrail
      Contact( #T1_ET60 )
      wire#w1
      Contact( #NXT_Avance_S4 )
      Contact( #PTF_Sal_M4 )
      wire#w2
      Contact( #PosTR_E2 )
      Contact( #EstadoZona.Marcha_CBx )
      I_Contact( #EstadoVI.Error_Mx )
      I_Contact( #EstadoZona.Manual_CBx )
      wire#w7
      Contact( #ok_tension )
      Coil( "DB1_SalidasExterioresDeMesa".Mesa[#Mesa].Avanzar_E2E4 )
   END_RUNG
   RUNG wire#w1
      I_Contact( #pHsMx )
   END_RUNG wire#w2
   RUNG wire#powerrail
      Contact( #T1_ET80 )
      wire#w3
      Contact( #NXT_Avance_S2 )
      Contact( #PTF_Sal_M2 )
   END_RUNG wire#w2
   RUNG wire#w3
      I_Contact( #pHsMx )
   END_RUNG wire#w2
   RUNG wire#powerrail
      Contact( #T1_ET20 )
      I_Contact( #tmp_pHs_E2_Q )
   END_RUNG wire#w2
   RUNG wire#powerrail
      Contact( #T1_ET21 )
      wire#w4
      Contact( #O_Sal_S4 )
      wire#w5
      Contact( #PTF_Sal_M4 )
   END_RUNG wire#w2
   RUNG wire#powerrail
      Contact( #T1_ET02 )
   END_RUNG wire#w4
   RUNG wire#w4
      Contact( #O_Bloqueo )
      wire#w6
      Contact( #Mx_FlujoPrin_S4 )
   END_RUNG wire#w5
   RUNG wire#w4
      Contact( #O_Vaciar )
   END_RUNG wire#w6
   RUNG wire#powerrail
      I_Contact( #Termico_24 )
      Contact( #EstadoZona.Rearme_CBx )
   END_RUNG wire#w7
   // the same network as SCL:
   "DB1_SalidasExterioresDeMesa".Mesa[#Mesa].Avanzar_E2E4 := ((((#T1_ET60 AND ((#NXT_Avance_S4 AND #PTF_Sal_M4) OR NOT #pHsMx)) OR (#T1_ET80 AND ((#NXT_Avance_S2 AND #PTF_Sal_M2) OR NOT #pHsMx)) OR (#T1_ET20 AND NOT #tmp_pHs_E2_Q) OR ((#T1_ET21 OR #T1_ET02) AND (#O_Sal_S4 OR ((#O_Bloqueo OR #O_Vaciar) AND #Mx_FlujoPrin_S4)) AND #PTF_Sal_M4)) AND #PosTR_E2 AND #EstadoZona.Marcha_CBx AND NOT #EstadoVI.Error_Mx AND NOT #EstadoZona.Manual_CBx) OR (NOT #Termico_24 AND #EstadoZona.Rearme_CBx)) AND #ok_tension;
END_REGION

REGION Network 65: invertir sentido de giro
   RUNG wire#powerrail
      Contact( #T1_ET80 )
      Contact( #NXT_Avance_S2 )
      Contact( #EstadoZona.Marcha_CBx )
      I_Contact( #EstadoVI.Error_Mx )
      I_Contact( #EstadoZona.Manual_CBx )
      Coil( #Inv_sentido_24 )
   END_RUNG
   // the same network as SCL:
   #Inv_sentido_24 := #T1_ET80 AND #NXT_Avance_S2 AND #EstadoZona.Marcha_CBx AND NOT #EstadoVI.Error_Mx AND NOT #EstadoZona.Manual_CBx;
END_REGION

REGION Network 66: #MA_AV_13_T_MX
   // Dani Palacios: en etapa 50 se deja que avance si no fotocelula. Es para 
   // asegurar 
   // que escribe la orden en el fifo y la puede leer el siguiente
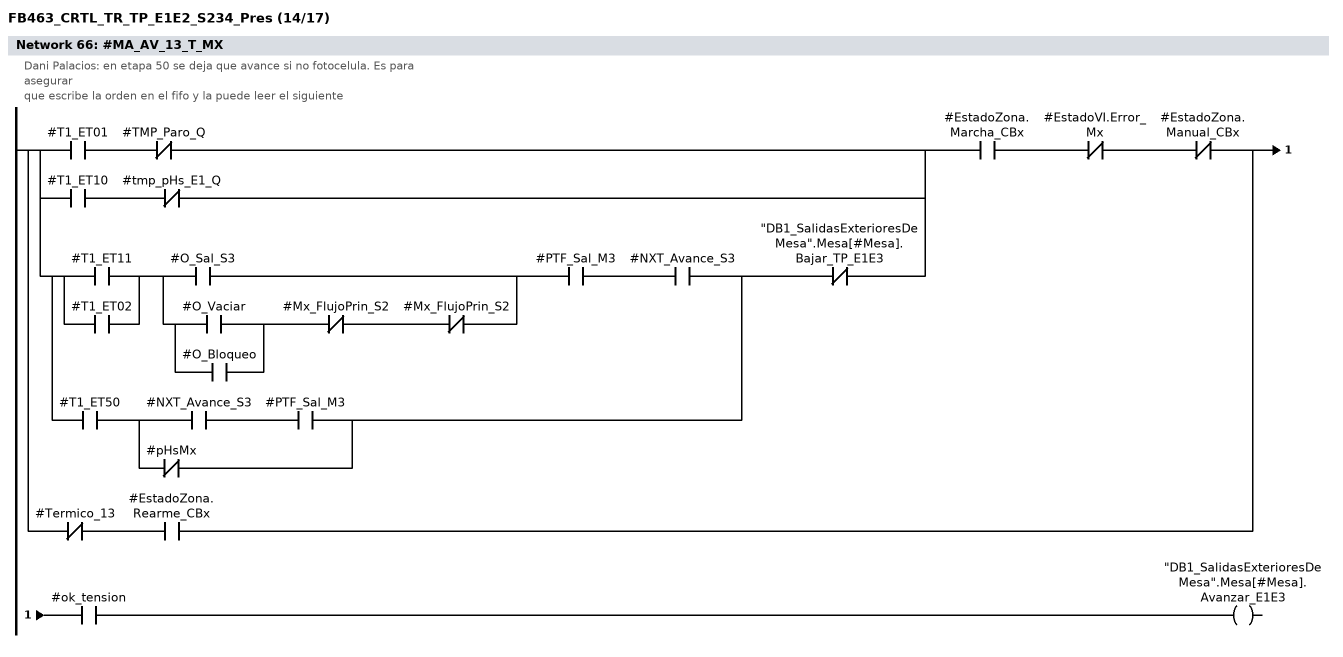
   RUNG wire#powerrail
      Contact( #T1_ET01 )
      I_Contact( #TMP_Paro_Q )
      wire#w1
      Contact( #EstadoZona.Marcha_CBx )
      I_Contact( #EstadoVI.Error_Mx )
      I_Contact( #EstadoZona.Manual_CBx )
      wire#w7
      Contact( #ok_tension )
      Coil( "DB1_SalidasExterioresDeMesa".Mesa[#Mesa].Avanzar_E1E3 )
   END_RUNG
   RUNG wire#powerrail
      Contact( #T1_ET10 )
      I_Contact( #tmp_pHs_E1_Q )
   END_RUNG wire#w1
   RUNG wire#powerrail
      Contact( #T1_ET11 )
      wire#w2
      Contact( #O_Sal_S3 )
      wire#w3
      Contact( #PTF_Sal_M3 )
      Contact( #NXT_Avance_S3 )
      wire#w5
      I_Contact( "DB1_SalidasExterioresDeMesa".Mesa[#Mesa].Bajar_TP_E1E3 )
   END_RUNG wire#w1
   RUNG wire#powerrail
      Contact( #T1_ET02 )
   END_RUNG wire#w2
   RUNG wire#w2
      Contact( #O_Vaciar )
      wire#w4
      I_Contact( #Mx_FlujoPrin_S2 )
      I_Contact( #Mx_FlujoPrin_S2 )
   END_RUNG wire#w3
   RUNG wire#w2
      Contact( #O_Bloqueo )
   END_RUNG wire#w4
   RUNG wire#powerrail
      Contact( #T1_ET50 )
      wire#w6
      Contact( #NXT_Avance_S3 )
      Contact( #PTF_Sal_M3 )
   END_RUNG wire#w5
   RUNG wire#w6
      I_Contact( #pHsMx )
   END_RUNG wire#w5
   RUNG wire#powerrail
      I_Contact( #Termico_13 )
      Contact( #EstadoZona.Rearme_CBx )
   END_RUNG wire#w7
   // the same network as SCL:
   "DB1_SalidasExterioresDeMesa".Mesa[#Mesa].Avanzar_E1E3 := ((((#T1_ET01 AND NOT #TMP_Paro_Q) OR (#T1_ET10 AND NOT #tmp_pHs_E1_Q) OR ((((#T1_ET11 OR #T1_ET02) AND (#O_Sal_S3 OR ((#O_Vaciar OR #O_Bloqueo) AND NOT #Mx_FlujoPrin_S2 AND NOT #Mx_FlujoPrin_S2)) AND #PTF_Sal_M3 AND #NXT_Avance_S3) OR (#T1_ET50 AND ((#NXT_Avance_S3 AND #PTF_Sal_M3) OR NOT #pHsMx))) AND NOT "DB1_SalidasExterioresDeMesa".Mesa[#Mesa].Bajar_TP_E1E3)) AND #EstadoZona.Marcha_CBx AND NOT #EstadoVI.Error_Mx AND NOT #EstadoZona.Manual_CBx) OR (NOT #Termico_13 AND #EstadoZona.Rearme_CBx)) AND #ok_tension;
END_REGION

REGION Network 67: PASAR ETIQUETA JDT
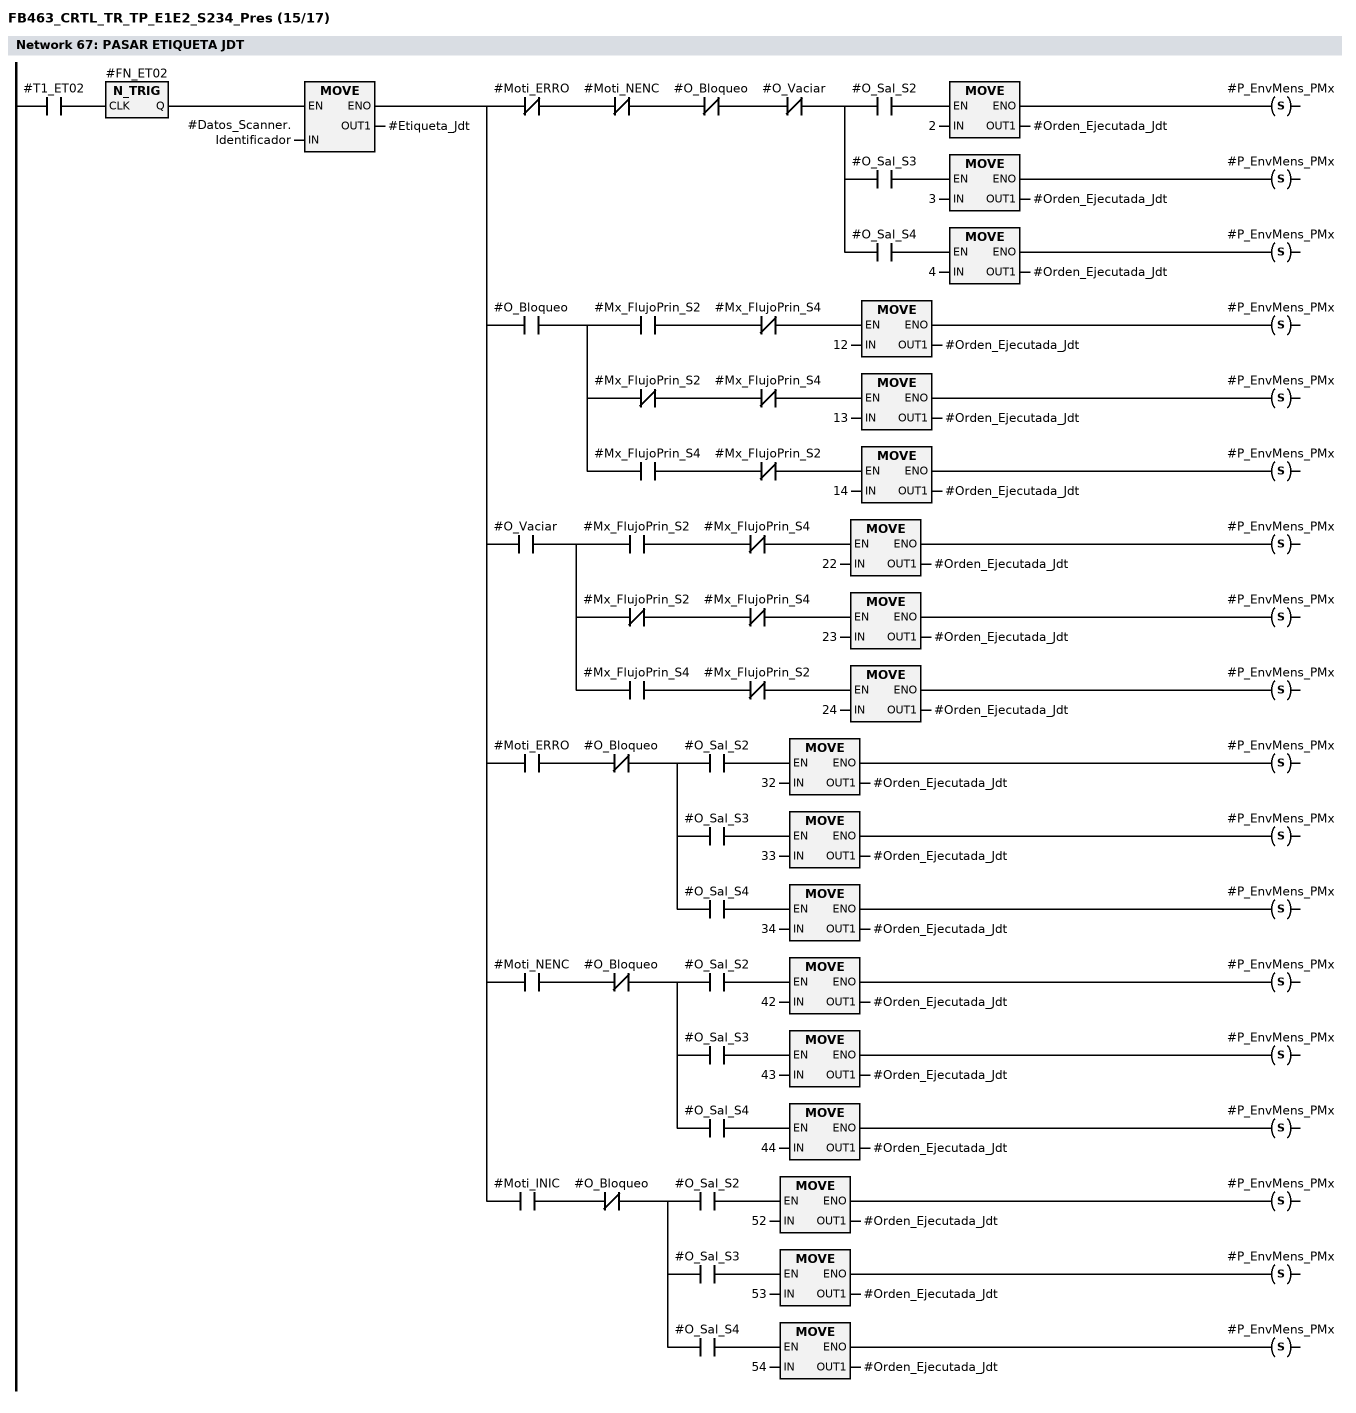
   RUNG wire#powerrail
      Contact( #T1_ET02 )
      N_Trig( #FN_ET02 )
      { S7_GenerateENO := "TRUE" } Move(in := #Datos_Scanner.Identificador, out1 => #Etiqueta_Jdt)
      wire#w1
      I_Contact( #Moti_ERRO )
      I_Contact( #Moti_NENC )
      I_Contact( #O_Bloqueo )
      I_Contact( #O_Vaciar )
      wire#w2
      Contact( #O_Sal_S2 )
      { S7_GenerateENO := "TRUE" } Move(in := 2, out1 => #Orden_Ejecutada_Jdt)
      S_Coil( #P_EnvMens_PMx )
   END_RUNG
   RUNG wire#w2
      Contact( #O_Sal_S3 )
      { S7_GenerateENO := "TRUE" } Move(in := 3, out1 => #Orden_Ejecutada_Jdt)
      S_Coil( #P_EnvMens_PMx )
   END_RUNG
   RUNG wire#w2
      Contact( #O_Sal_S4 )
      { S7_GenerateENO := "TRUE" } Move(in := 4, out1 => #Orden_Ejecutada_Jdt)
      S_Coil( #P_EnvMens_PMx )
   END_RUNG
   RUNG wire#w1
      Contact( #O_Bloqueo )
      wire#w3
      Contact( #Mx_FlujoPrin_S2 )
      I_Contact( #Mx_FlujoPrin_S4 )
      { S7_GenerateENO := "TRUE" } Move(in := 12, out1 => #Orden_Ejecutada_Jdt)
      S_Coil( #P_EnvMens_PMx )
   END_RUNG
   RUNG wire#w3
      I_Contact( #Mx_FlujoPrin_S2 )
      I_Contact( #Mx_FlujoPrin_S4 )
      { S7_GenerateENO := "TRUE" } Move(in := 13, out1 => #Orden_Ejecutada_Jdt)
      S_Coil( #P_EnvMens_PMx )
   END_RUNG
   RUNG wire#w3
      Contact( #Mx_FlujoPrin_S4 )
      I_Contact( #Mx_FlujoPrin_S2 )
      { S7_GenerateENO := "TRUE" } Move(in := 14, out1 => #Orden_Ejecutada_Jdt)
      S_Coil( #P_EnvMens_PMx )
   END_RUNG
   RUNG wire#w1
      Contact( #O_Vaciar )
      wire#w4
      Contact( #Mx_FlujoPrin_S2 )
      I_Contact( #Mx_FlujoPrin_S4 )
      { S7_GenerateENO := "TRUE" } Move(in := 22, out1 => #Orden_Ejecutada_Jdt)
      S_Coil( #P_EnvMens_PMx )
   END_RUNG
   RUNG wire#w4
      I_Contact( #Mx_FlujoPrin_S2 )
      I_Contact( #Mx_FlujoPrin_S4 )
      { S7_GenerateENO := "TRUE" } Move(in := 23, out1 => #Orden_Ejecutada_Jdt)
      S_Coil( #P_EnvMens_PMx )
   END_RUNG
   RUNG wire#w4
      Contact( #Mx_FlujoPrin_S4 )
      I_Contact( #Mx_FlujoPrin_S2 )
      { S7_GenerateENO := "TRUE" } Move(in := 24, out1 => #Orden_Ejecutada_Jdt)
      S_Coil( #P_EnvMens_PMx )
   END_RUNG
   RUNG wire#w1
      Contact( #Moti_ERRO )
      I_Contact( #O_Bloqueo )
      wire#w5
      Contact( #O_Sal_S2 )
      { S7_GenerateENO := "TRUE" } Move(in := 32, out1 => #Orden_Ejecutada_Jdt)
      S_Coil( #P_EnvMens_PMx )
   END_RUNG
   RUNG wire#w5
      Contact( #O_Sal_S3 )
      { S7_GenerateENO := "TRUE" } Move(in := 33, out1 => #Orden_Ejecutada_Jdt)
      S_Coil( #P_EnvMens_PMx )
   END_RUNG
   RUNG wire#w5
      Contact( #O_Sal_S4 )
      { S7_GenerateENO := "TRUE" } Move(in := 34, out1 => #Orden_Ejecutada_Jdt)
      S_Coil( #P_EnvMens_PMx )
   END_RUNG
   RUNG wire#w1
      Contact( #Moti_NENC )
      I_Contact( #O_Bloqueo )
      wire#w6
      Contact( #O_Sal_S2 )
      { S7_GenerateENO := "TRUE" } Move(in := 42, out1 => #Orden_Ejecutada_Jdt)
      S_Coil( #P_EnvMens_PMx )
   END_RUNG
   RUNG wire#w6
      Contact( #O_Sal_S3 )
      { S7_GenerateENO := "TRUE" } Move(in := 43, out1 => #Orden_Ejecutada_Jdt)
      S_Coil( #P_EnvMens_PMx )
   END_RUNG
   RUNG wire#w6
      Contact( #O_Sal_S4 )
      { S7_GenerateENO := "TRUE" } Move(in := 44, out1 => #Orden_Ejecutada_Jdt)
      S_Coil( #P_EnvMens_PMx )
   END_RUNG
   RUNG wire#w1
      Contact( #Moti_INIC )
      I_Contact( #O_Bloqueo )
      wire#w7
      Contact( #O_Sal_S2 )
      { S7_GenerateENO := "TRUE" } Move(in := 52, out1 => #Orden_Ejecutada_Jdt)
      S_Coil( #P_EnvMens_PMx )
   END_RUNG
   RUNG wire#w7
      Contact( #O_Sal_S3 )
      { S7_GenerateENO := "TRUE" } Move(in := 53, out1 => #Orden_Ejecutada_Jdt)
      S_Coil( #P_EnvMens_PMx )
   END_RUNG
   RUNG wire#w7
      Contact( #O_Sal_S4 )
      { S7_GenerateENO := "TRUE" } Move(in := 54, out1 => #Orden_Ejecutada_Jdt)
      S_Coil( #P_EnvMens_PMx )
   END_RUNG
   // the same network as SCL:
   // ENO of a box is taken as its EN; it also drops when the box reports an error
   #_w1 := NOT #T1_ET02 AND #FN_ET02;   // falling edge
   #FN_ET02 := #T1_ET02;
   IF #_w1 THEN #Etiqueta_Jdt := #Datos_Scanner.Identificador; END_IF;
   #_w2 := #_w1 AND NOT #Moti_ERRO AND NOT #Moti_NENC AND NOT #O_Bloqueo AND NOT #O_Vaciar;
   IF #_w2 AND #O_Sal_S2 THEN
       #Orden_Ejecutada_Jdt := 2;
       #P_EnvMens_PMx := TRUE;
   END_IF;
   IF #_w2 AND #O_Sal_S3 THEN
       #Orden_Ejecutada_Jdt := 3;
       #P_EnvMens_PMx := TRUE;
   END_IF;
   IF #_w2 AND #O_Sal_S4 THEN
       #Orden_Ejecutada_Jdt := 4;
       #P_EnvMens_PMx := TRUE;
   END_IF;
   #_w3 := #_w1 AND #O_Bloqueo;
   IF #_w3 AND #Mx_FlujoPrin_S2 AND NOT #Mx_FlujoPrin_S4 THEN
       #Orden_Ejecutada_Jdt := 12;
       #P_EnvMens_PMx := TRUE;
   END_IF;
   IF #_w3 AND NOT #Mx_FlujoPrin_S2 AND NOT #Mx_FlujoPrin_S4 THEN
       #Orden_Ejecutada_Jdt := 13;
       #P_EnvMens_PMx := TRUE;
   END_IF;
   IF #_w3 AND #Mx_FlujoPrin_S4 AND NOT #Mx_FlujoPrin_S2 THEN
       #Orden_Ejecutada_Jdt := 14;
       #P_EnvMens_PMx := TRUE;
   END_IF;
   #_w4 := #_w1 AND #O_Vaciar;
   IF #_w4 AND #Mx_FlujoPrin_S2 AND NOT #Mx_FlujoPrin_S4 THEN
       #Orden_Ejecutada_Jdt := 22;
       #P_EnvMens_PMx := TRUE;
   END_IF;
   IF #_w4 AND NOT #Mx_FlujoPrin_S2 AND NOT #Mx_FlujoPrin_S4 THEN
       #Orden_Ejecutada_Jdt := 23;
       #P_EnvMens_PMx := TRUE;
   END_IF;
   IF #_w4 AND #Mx_FlujoPrin_S4 AND NOT #Mx_FlujoPrin_S2 THEN
       #Orden_Ejecutada_Jdt := 24;
       #P_EnvMens_PMx := TRUE;
   END_IF;
   #_w5 := #_w1 AND #Moti_ERRO AND NOT #O_Bloqueo;
   IF #_w5 AND #O_Sal_S2 THEN
       #Orden_Ejecutada_Jdt := 32;
       #P_EnvMens_PMx := TRUE;
   END_IF;
   IF #_w5 AND #O_Sal_S3 THEN
       #Orden_Ejecutada_Jdt := 33;
       #P_EnvMens_PMx := TRUE;
   END_IF;
   IF #_w5 AND #O_Sal_S4 THEN
       #Orden_Ejecutada_Jdt := 34;
       #P_EnvMens_PMx := TRUE;
   END_IF;
   #_w6 := #_w1 AND #Moti_NENC AND NOT #O_Bloqueo;
   IF #_w6 AND #O_Sal_S2 THEN
       #Orden_Ejecutada_Jdt := 42;
       #P_EnvMens_PMx := TRUE;
   END_IF;
   IF #_w6 AND #O_Sal_S3 THEN
       #Orden_Ejecutada_Jdt := 43;
       #P_EnvMens_PMx := TRUE;
   END_IF;
   IF #_w6 AND #O_Sal_S4 THEN
       #Orden_Ejecutada_Jdt := 44;
       #P_EnvMens_PMx := TRUE;
   END_IF;
   #_w7 := #_w1 AND #Moti_INIC AND NOT #O_Bloqueo;
   IF #_w7 AND #O_Sal_S2 THEN
       #Orden_Ejecutada_Jdt := 52;
       #P_EnvMens_PMx := TRUE;
   END_IF;
   IF #_w7 AND #O_Sal_S3 THEN
       #Orden_Ejecutada_Jdt := 53;
       #P_EnvMens_PMx := TRUE;
   END_IF;
   IF #_w7 AND #O_Sal_S4 THEN
       #Orden_Ejecutada_Jdt := 54;
       #P_EnvMens_PMx := TRUE;
   END_IF;
END_REGION

REGION Network 68: R presencia JDT
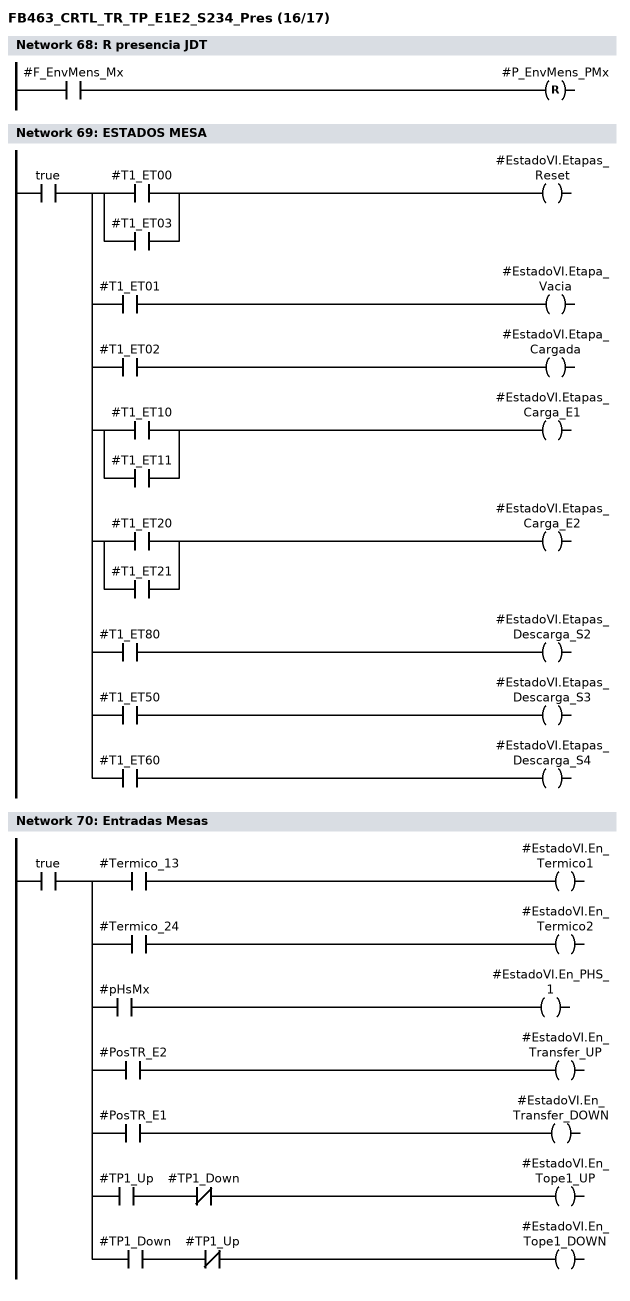
   RUNG wire#powerrail
      Contact( #F_EnvMens_Mx )
      R_Coil( #P_EnvMens_PMx )
   END_RUNG
   // the same network as SCL:
   IF #F_EnvMens_Mx THEN #P_EnvMens_PMx := FALSE; END_IF;
END_REGION

REGION Network 69: ESTADOS MESA
   RUNG wire#powerrail
      Contact( true )
      wire#w1
      Contact( #T1_ET00 )
      wire#w2
      Coil( #EstadoVI.Etapas_Reset )
   END_RUNG
   RUNG wire#w1
      Contact( #T1_ET03 )
   END_RUNG wire#w2
   RUNG wire#w1
      Contact( #T1_ET01 )
      Coil( #EstadoVI.Etapa_Vacia )
   END_RUNG
   RUNG wire#w1
      Contact( #T1_ET02 )
      Coil( #EstadoVI.Etapa_Cargada )
   END_RUNG
   RUNG wire#w1
      Contact( #T1_ET10 )
      wire#w3
      Coil( #EstadoVI.Etapas_Carga_E1 )
   END_RUNG
   RUNG wire#w1
      Contact( #T1_ET11 )
   END_RUNG wire#w3
   RUNG wire#w1
      Contact( #T1_ET20 )
      wire#w4
      Coil( #EstadoVI.Etapas_Carga_E2 )
   END_RUNG
   RUNG wire#w1
      Contact( #T1_ET21 )
   END_RUNG wire#w4
   RUNG wire#w1
      Contact( #T1_ET80 )
      Coil( #EstadoVI.Etapas_Descarga_S2 )
   END_RUNG
   RUNG wire#w1
      Contact( #T1_ET50 )
      Coil( #EstadoVI.Etapas_Descarga_S3 )
   END_RUNG
   RUNG wire#w1
      Contact( #T1_ET60 )
      Coil( #EstadoVI.Etapas_Descarga_S4 )
   END_RUNG
   // the same network as SCL:
   #EstadoVI.Etapas_Reset := true AND (#T1_ET00 OR #T1_ET03);
   #EstadoVI.Etapa_Vacia := true AND #T1_ET01;
   #EstadoVI.Etapa_Cargada := true AND #T1_ET02;
   #EstadoVI.Etapas_Carga_E1 := true AND (#T1_ET10 OR #T1_ET11);
   #EstadoVI.Etapas_Carga_E2 := true AND (#T1_ET20 OR #T1_ET21);
   #EstadoVI.Etapas_Descarga_S2 := true AND #T1_ET80;
   #EstadoVI.Etapas_Descarga_S3 := true AND #T1_ET50;
   #EstadoVI.Etapas_Descarga_S4 := true AND #T1_ET60;
END_REGION

REGION Network 70: Entradas Mesas
   RUNG wire#powerrail
      Contact( true )
      wire#w1
      Contact( #Termico_13 )
      Coil( #EstadoVI.En_Termico1 )
   END_RUNG
   RUNG wire#w1
      Contact( #Termico_24 )
      Coil( #EstadoVI.En_Termico2 )
   END_RUNG
   RUNG wire#w1
      Contact( #pHsMx )
      Coil( #EstadoVI.En_PHS_1 )
   END_RUNG
   RUNG wire#w1
      Contact( #PosTR_E2 )
      Coil( #EstadoVI.En_Transfer_UP )
   END_RUNG
   RUNG wire#w1
      Contact( #PosTR_E1 )
      Coil( #EstadoVI.En_Transfer_DOWN )
   END_RUNG
   RUNG wire#w1
      Contact( #TP1_Up )
      I_Contact( #TP1_Down )
      Coil( #EstadoVI.En_Tope1_UP )
   END_RUNG
   RUNG wire#w1
      Contact( #TP1_Down )
      I_Contact( #TP1_Up )
      Coil( #EstadoVI.En_Tope1_DOWN )
   END_RUNG
   // the same network as SCL:
   #EstadoVI.En_Termico1 := true AND #Termico_13;
   #EstadoVI.En_Termico2 := true AND #Termico_24;
   #EstadoVI.En_PHS_1 := true AND #pHsMx;
   #EstadoVI.En_Transfer_UP := true AND #PosTR_E2;
   #EstadoVI.En_Transfer_DOWN := true AND #PosTR_E1;
   #EstadoVI.En_Tope1_UP := true AND #TP1_Up AND NOT #TP1_Down;
   #EstadoVI.En_Tope1_DOWN := true AND #TP1_Down AND NOT #TP1_Up;
END_REGION

REGION Network 71: Salidas Mesas
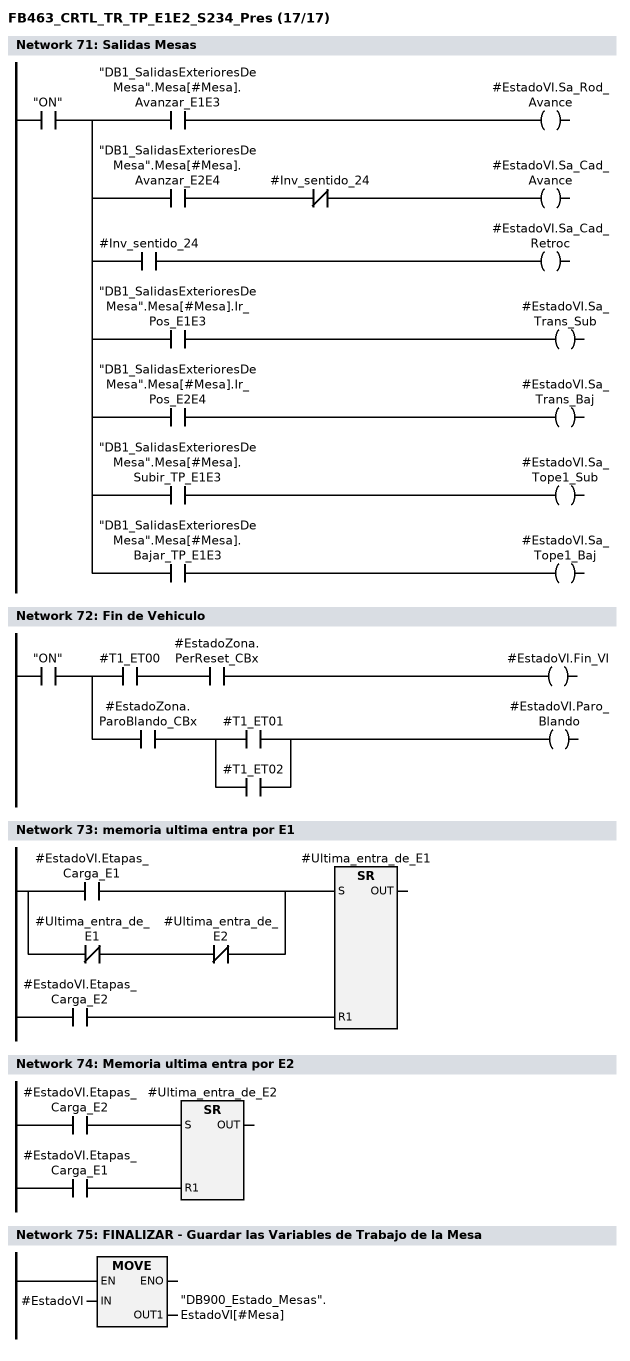
   RUNG wire#powerrail
      Contact( "ON" )
      wire#w1
      Contact( "DB1_SalidasExterioresDeMesa".Mesa[#Mesa].Avanzar_E1E3 )
      Coil( #EstadoVI.Sa_Rod_Avance )
   END_RUNG
   RUNG wire#w1
      Contact( "DB1_SalidasExterioresDeMesa".Mesa[#Mesa].Avanzar_E2E4 )
      I_Contact( #Inv_sentido_24 )
      Coil( #EstadoVI.Sa_Cad_Avance )
   END_RUNG
   RUNG wire#w1
      Contact( #Inv_sentido_24 )
      Coil( #EstadoVI.Sa_Cad_Retroc )
   END_RUNG
   RUNG wire#w1
      Contact( "DB1_SalidasExterioresDeMesa".Mesa[#Mesa].Ir_Pos_E1E3 )
      Coil( #EstadoVI.Sa_Trans_Sub )
   END_RUNG
   RUNG wire#w1
      Contact( "DB1_SalidasExterioresDeMesa".Mesa[#Mesa].Ir_Pos_E2E4 )
      Coil( #EstadoVI.Sa_Trans_Baj )
   END_RUNG
   RUNG wire#w1
      Contact( "DB1_SalidasExterioresDeMesa".Mesa[#Mesa].Subir_TP_E1E3 )
      Coil( #EstadoVI.Sa_Tope1_Sub )
   END_RUNG
   RUNG wire#w1
      Contact( "DB1_SalidasExterioresDeMesa".Mesa[#Mesa].Bajar_TP_E1E3 )
      Coil( #EstadoVI.Sa_Tope1_Baj )
   END_RUNG
   // the same network as SCL:
   #EstadoVI.Sa_Rod_Avance := "ON" AND "DB1_SalidasExterioresDeMesa".Mesa[#Mesa].Avanzar_E1E3;
   #EstadoVI.Sa_Cad_Avance := "ON" AND "DB1_SalidasExterioresDeMesa".Mesa[#Mesa].Avanzar_E2E4 AND NOT #Inv_sentido_24;
   #EstadoVI.Sa_Cad_Retroc := "ON" AND #Inv_sentido_24;
   #EstadoVI.Sa_Trans_Sub := "ON" AND "DB1_SalidasExterioresDeMesa".Mesa[#Mesa].Ir_Pos_E1E3;
   #EstadoVI.Sa_Trans_Baj := "ON" AND "DB1_SalidasExterioresDeMesa".Mesa[#Mesa].Ir_Pos_E2E4;
   #EstadoVI.Sa_Tope1_Sub := "ON" AND "DB1_SalidasExterioresDeMesa".Mesa[#Mesa].Subir_TP_E1E3;
   #EstadoVI.Sa_Tope1_Baj := "ON" AND "DB1_SalidasExterioresDeMesa".Mesa[#Mesa].Bajar_TP_E1E3;
END_REGION

REGION Network 72: Fin de Vehiculo
   RUNG wire#powerrail
      Contact( "ON" )
      wire#w1
      Contact( #T1_ET00 )
      Contact( #EstadoZona.PerReset_CBx )
      Coil( #EstadoVI.Fin_VI )
   END_RUNG
   RUNG wire#w1
      Contact( #EstadoZona.ParoBlando_CBx )
      wire#w2
      Contact( #T1_ET01 )
      wire#w3
      Coil( #EstadoVI.Paro_Blando )
   END_RUNG
   RUNG wire#w2
      Contact( #T1_ET02 )
   END_RUNG wire#w3
   // the same network as SCL:
   #EstadoVI.Fin_VI := "ON" AND #T1_ET00 AND #EstadoZona.PerReset_CBx;
   #EstadoVI.Paro_Blando := "ON" AND #EstadoZona.ParoBlando_CBx AND (#T1_ET01 OR #T1_ET02);
END_REGION

REGION Network 73: memoria ultima entra por E1
   RUNG wire#powerrail
      Contact( #EstadoVI.Etapas_Carga_E1 )
      wire#w1
      S_SR(operand := #Ultima_entra_de_E1, r1 := wire#w2)
   END_RUNG
   RUNG wire#powerrail
      I_Contact( #Ultima_entra_de_E1 )
      I_Contact( #Ultima_entra_de_E2 )
   END_RUNG wire#w1
   RUNG wire#powerrail
      Contact( #EstadoVI.Etapas_Carga_E2 )
   END_RUNG wire#w2
   // the same network as SCL:
   IF #EstadoVI.Etapas_Carga_E1 OR (NOT #Ultima_entra_de_E1 AND NOT #Ultima_entra_de_E2) THEN
       #Ultima_entra_de_E1 := TRUE;   // SR flip-flop
   END_IF;
   IF #EstadoVI.Etapas_Carga_E2 THEN #Ultima_entra_de_E1 := FALSE; END_IF;
END_REGION

REGION Network 74: Memoria ultima entra por E2
   RUNG wire#powerrail
      Contact( #EstadoVI.Etapas_Carga_E2 )
      S_SR(operand := #Ultima_entra_de_E2, r1 := wire#w1)
   END_RUNG
   RUNG wire#powerrail
      Contact( #EstadoVI.Etapas_Carga_E1 )
   END_RUNG wire#w1
   // the same network as SCL:
   IF #EstadoVI.Etapas_Carga_E2 THEN
       #Ultima_entra_de_E2 := TRUE;   // SR flip-flop
   END_IF;
   IF #EstadoVI.Etapas_Carga_E1 THEN #Ultima_entra_de_E2 := FALSE; END_IF;
END_REGION

REGION Network 75: FINALIZAR - Guardar las Variables de Trabajo de la Mesa
   RUNG wire#powerrail
      Move(in := #EstadoVI, out1 => "DB900_Estado_Mesas".EstadoVI[#Mesa])
   END_RUNG
   // the same network as SCL:
   "DB900_Estado_Mesas".EstadoVI[#Mesa] := #EstadoVI;
END_REGION
END_FUNCTION_BLOCK
